// TwinCAT 3 PLC project PLC1
// Title: XPlanar Example Project
// Company: Beckhoff Automation LLC
// ProjectVersion: 1.0.0
// ProgramVersion: 3.1.4023.0
// libraries:
//   SPT Base Types, * (Beckhoff Automation LLC)
//   SPT Event Logger, * (Beckhoff Automation LLC)
//   SPT_XPlanar, * (Beckhoff Automation LLC)
//   Tc2_EtherCAT, * (Beckhoff Automation GmbH)
//   Tc2_Math, * (Beckhoff Automation GmbH)
//   Tc2_Standard, * (Beckhoff Automation GmbH)
//   Tc2_System, * (Beckhoff Automation GmbH)
//   Tc3_EventLogger, * (Beckhoff Automation GmbH)
//   Tc3_Module, * (Beckhoff Automation GmbH)
//   Tc3_PackML_V2, * (Beckhoff Automation GmbH)
//   Tc3_XPlanarUtility, * (Beckhoff Automation GmbH & Co. KG)
//   Tc3_Mc3PlanarMotion,newest,Beckhoff Automation GmbH
//   Tc3_Physics,newest,Beckhoff Automation GmbH
//   Tc3_XPlanarStandard,newest,Beckhoff Automation GmbH
//   VisuSymbols,3.5.10.0,System
// project tree:
//   DUTS/ ST_StationPosition.TcDUT, ST_VisMover.TcDUT, ST_VisStationData.TcDUT
//   / GlobalTextList.TcGTLO, MAIN.TcPOU, NextMinorStep.TcPOU, NextStep.TcPOU, PlcTask.TcTTO (not stored), StationList_TextList.TcTLO (not stored), Visualization Manager.TcVMO (not stored)
//   GVL/ GVL_Xplanar.TcGVL
//   Logic/Initialize/ FB_BasicInitialization.TcPOU, FB_MoverList.TcPOU
//   Machine/EquipmentModules/CustomStations/ FB_DecisionStation.TcPOU, FB_SpinStation.TcPOU
//   Machine/EquipmentModules/ FB_XPlanar_EM.TcPOU
//   Machine/ FB_Machine.TcPOU
//   Machine/VISUs/VisuOjects/ V_Control_Xplanar.TcVIS, V_MachineModule.TcVIS, V_Module.TcVIS (not stored), V_Mover.TcVIS (not stored), V_RotaryAxis.TcVIS (not stored), V_Station.TcVIS
//   Machine/VISUs/ V_Main.TcVIS
// real-time tasks:
//   TASK PlcTask: cycle T#10ms, priority 20, ADS port 350
//   TASK MC-Task (MET): cycle T#2ms, priority 7, ADS port 357
//   TASK MC-Task (MPT): cycle T#10ms, priority 8, ADS port 358
//   TASK Job Task: cycle default, priority 9
//   TASK XPlanar Task9: cycle T#250us, priority 1, ADS port 351
//   TASK XPlanar Task10: cycle T#250us, priority 2, ADS port 352
//   TASK XPlanar Task11: cycle T#250us, priority 3, ADS port 353
//   TASK XPlanar Task12: cycle T#250us, priority 4, ADS port 354
//   TASK XPlanar Task13: cycle T#250us, priority 5, ADS port 355
//   TASK XPlanar Task14: cycle T#250us, priority 6, ADS port 356
//   TASK XPlanar Task15: cycle T#250us, priority 10, ADS port 359
// variable links:
//   XPlanar MC Project/Axes/Mover4220_1 <-> TcCOM Objects/XPlanar/Mover4220_1
//     McToIo/STD <-> InputsFromNC3/NC3ToHW
//   XPlanar MC Project/Axes/Mover4220_10 <-> TcCOM Objects/XPlanar/Mover4220_10
//     McToIo/STD <-> InputsFromNC3/NC3ToHW
//   XPlanar MC Project/Axes/Mover4220_12 <-> TcCOM Objects/XPlanar/Mover4220_12
//     McToIo/STD <-> InputsFromNC3/NC3ToHW
//   XPlanar MC Project/Axes/Mover4220_13 <-> TcCOM Objects/XPlanar/Mover4220_13
//     IoToMc/STD <-> OutputsToNC3/HWToNC3
//   XPlanar MC Project/Axes/Mover4220_14 <-> TcCOM Objects/XPlanar/Mover4220_14
//     IoToMc/STD <-> OutputsToNC3/HWToNC3
//   XPlanar MC Project/Axes/Mover4220_15 <-> TcCOM Objects/XPlanar/Mover4220_15
//     IoToMc/STD <-> OutputsToNC3/HWToNC3
//     McToIo/STD <-> InputsFromNC3/NC3ToHW
//   XPlanar MC Project/Axes/Mover4220_17 <-> TcCOM Objects/XPlanar/Mover4220_17
//     IoToMc/STD <-> OutputsToNC3/HWToNC3
//     McToIo/STD <-> InputsFromNC3/NC3ToHW
//   XPlanar MC Project/Axes/Mover4220_18 <-> TcCOM Objects/XPlanar/Mover4220_18
//     IoToMc/STD <-> OutputsToNC3/HWToNC3
//     McToIo/STD <-> InputsFromNC3/NC3ToHW
//   XPlanar MC Project/Axes/Mover4220_19 <-> TcCOM Objects/XPlanar/Mover4220_19
//     McToIo/STD <-> InputsFromNC3/NC3ToHW
//   XPlanar MC Project/Axes/Mover4220_2 <-> TcCOM Objects/XPlanar/Mover4220_2
//     McToIo/STD <-> InputsFromNC3/NC3ToHW
//   XPlanar MC Project/Axes/Mover4220_3 <-> TcCOM Objects/XPlanar/Mover4220_3
//     IoToMc/STD <-> OutputsToNC3/HWToNC3
//   XPlanar MC Project/Axes/Mover4220_4 <-> TcCOM Objects/XPlanar/Mover4220_4
//     IoToMc/STD <-> OutputsToNC3/HWToNC3
//   XPlanar MC Project/Axes/Mover4220_5 <-> TcCOM Objects/XPlanar/Mover4220_5
//     IoToMc/STD <-> OutputsToNC3/HWToNC3
//     McToIo/STD <-> InputsFromNC3/NC3ToHW
//   XPlanar MC Project/Axes/Mover4220_6 <-> TcCOM Objects/XPlanar/Mover4220_6
//     McToIo/STD <-> InputsFromNC3/NC3ToHW
//   XPlanar MC Project/Axes/Mover4220_7 <-> TcCOM Objects/XPlanar/Mover4220_7
//     IoToMc/STD <-> OutputsToNC3/HWToNC3
//     McToIo/STD <-> InputsFromNC3/NC3ToHW
//   XPlanar MC Project/Axes/Mover4220_9 <-> TcCOM Objects/XPlanar/Mover4220_9
//     IoToMc/STD <-> OutputsToNC3/HWToNC3
//     McToIo/STD <-> InputsFromNC3/NC3ToHW
//   PLC1/PLC1 Instance <-> XPlanar MC Project/Axes/Mover4220_1
//     PlcTask Inputs/MAIN.Machine.XPlanar.Movers[1]._Mover.stMoverRef.MCTOPLC/ACT <-> McToPlc/ACT
//     PlcTask Inputs/MAIN.Machine.XPlanar.Movers[1]._Mover.stMoverRef.MCTOPLC/COORDMODE <-> McToPlc/COORDMODE
//     PlcTask Inputs/MAIN.Machine.XPlanar.Movers[1]._Mover.stMoverRef.MCTOPLC/SET <-> McToPlc/SET
//     PlcTask Inputs/MAIN.Machine.XPlanar.Movers[1]._Mover.stMoverRef.MCTOPLC/SETONTRACK <-> McToPlc/SETONTRACK
//     PlcTask Inputs/MAIN.Machine.XPlanar.Movers[1]._Mover.stMoverRef.MCTOPLC/STD <-> McToPlc/STD
//     PlcTask Outputs/MAIN.Machine.XPlanar.Movers[1]._Mover.stMoverRef.PLCTOMC/STD <-> PlcToMc/STD
//   PLC1/PLC1 Instance <-> XPlanar MC Project/Axes/Mover4220_10
//     PlcTask Inputs/MAIN.Machine.XPlanar.Movers[10]._Mover.stMoverRef.MCTOPLC/ACT <-> McToPlc/ACT
//     PlcTask Inputs/MAIN.Machine.XPlanar.Movers[10]._Mover.stMoverRef.MCTOPLC/COORDMODE <-> McToPlc/COORDMODE
//     PlcTask Inputs/MAIN.Machine.XPlanar.Movers[10]._Mover.stMoverRef.MCTOPLC/SET <-> McToPlc/SET
//     PlcTask Inputs/MAIN.Machine.XPlanar.Movers[10]._Mover.stMoverRef.MCTOPLC/SETONTRACK <-> McToPlc/SETONTRACK
//     PlcTask Inputs/MAIN.Machine.XPlanar.Movers[10]._Mover.stMoverRef.MCTOPLC/STD <-> McToPlc/STD
//     PlcTask Outputs/MAIN.Machine.XPlanar.Movers[10]._Mover.stMoverRef.PLCTOMC/STD <-> PlcToMc/STD
//   PLC1/PLC1 Instance <-> XPlanar MC Project/Axes/Mover4220_11
//     PlcTask Inputs/MAIN.Machine.XPlanar.Movers[11]._Mover.stMoverRef.MCTOPLC/ACT <-> McToPlc/ACT
//     PlcTask Inputs/MAIN.Machine.XPlanar.Movers[11]._Mover.stMoverRef.MCTOPLC/COORDMODE <-> McToPlc/COORDMODE
//     PlcTask Inputs/MAIN.Machine.XPlanar.Movers[11]._Mover.stMoverRef.MCTOPLC/SET <-> McToPlc/SET
//     PlcTask Inputs/MAIN.Machine.XPlanar.Movers[11]._Mover.stMoverRef.MCTOPLC/SETONTRACK <-> McToPlc/SETONTRACK
//     PlcTask Inputs/MAIN.Machine.XPlanar.Movers[11]._Mover.stMoverRef.MCTOPLC/STD <-> McToPlc/STD
//     PlcTask Outputs/MAIN.Machine.XPlanar.Movers[11]._Mover.stMoverRef.PLCTOMC/STD <-> PlcToMc/STD
//   PLC1/PLC1 Instance <-> XPlanar MC Project/Axes/Mover4220_12
//     PlcTask Inputs/MAIN.Machine.XPlanar.Movers[12]._Mover.stMoverRef.MCTOPLC/ACT <-> McToPlc/ACT
//     PlcTask Inputs/MAIN.Machine.XPlanar.Movers[12]._Mover.stMoverRef.MCTOPLC/COORDMODE <-> McToPlc/COORDMODE
//     PlcTask Inputs/MAIN.Machine.XPlanar.Movers[12]._Mover.stMoverRef.MCTOPLC/SET <-> McToPlc/SET
//     PlcTask Inputs/MAIN.Machine.XPlanar.Movers[12]._Mover.stMoverRef.MCTOPLC/SETONTRACK <-> McToPlc/SETONTRACK
//     PlcTask Inputs/MAIN.Machine.XPlanar.Movers[12]._Mover.stMoverRef.MCTOPLC/STD <-> McToPlc/STD
//     PlcTask Outputs/MAIN.Machine.XPlanar.Movers[12]._Mover.stMoverRef.PLCTOMC/STD <-> PlcToMc/STD
//   PLC1/PLC1 Instance <-> XPlanar MC Project/Axes/Mover4220_13
//     PlcTask Inputs/MAIN.Machine.XPlanar.Movers[13]._Mover.stMoverRef.MCTOPLC/ACT <-> McToPlc/ACT
//     PlcTask Inputs/MAIN.Machine.XPlanar.Movers[13]._Mover.stMoverRef.MCTOPLC/COORDMODE <-> McToPlc/COORDMODE
//     PlcTask Inputs/MAIN.Machine.XPlanar.Movers[13]._Mover.stMoverRef.MCTOPLC/SET <-> McToPlc/SET
//     PlcTask Inputs/MAIN.Machine.XPlanar.Movers[13]._Mover.stMoverRef.MCTOPLC/SETONTRACK <-> McToPlc/SETONTRACK
//     PlcTask Inputs/MAIN.Machine.XPlanar.Movers[13]._Mover.stMoverRef.MCTOPLC/STD <-> McToPlc/STD
//     PlcTask Outputs/MAIN.Machine.XPlanar.Movers[13]._Mover.stMoverRef.PLCTOMC/STD <-> PlcToMc/STD
//   PLC1/PLC1 Instance <-> XPlanar MC Project/Axes/Mover4220_14
//     PlcTask Inputs/MAIN.Machine.XPlanar.Movers[14]._Mover.stMoverRef.MCTOPLC/ACT <-> McToPlc/ACT
//     PlcTask Inputs/MAIN.Machine.XPlanar.Movers[14]._Mover.stMoverRef.MCTOPLC/COORDMODE <-> McToPlc/COORDMODE
//     PlcTask Inputs/MAIN.Machine.XPlanar.Movers[14]._Mover.stMoverRef.MCTOPLC/SET <-> McToPlc/SET
//     PlcTask Inputs/MAIN.Machine.XPlanar.Movers[14]._Mover.stMoverRef.MCTOPLC/SETONTRACK <-> McToPlc/SETONTRACK
//     PlcTask Inputs/MAIN.Machine.XPlanar.Movers[14]._Mover.stMoverRef.MCTOPLC/STD <-> McToPlc/STD
//     PlcTask Outputs/MAIN.Machine.XPlanar.Movers[14]._Mover.stMoverRef.PLCTOMC/STD <-> PlcToMc/STD
//   PLC1/PLC1 Instance <-> XPlanar MC Project/Axes/Mover4220_15
//     PlcTask Inputs/MAIN.Machine.XPlanar.Movers[15]._Mover.stMoverRef.MCTOPLC/ACT <-> McToPlc/ACT
//     PlcTask Inputs/MAIN.Machine.XPlanar.Movers[15]._Mover.stMoverRef.MCTOPLC/COORDMODE <-> McToPlc/COORDMODE
//     PlcTask Inputs/MAIN.Machine.XPlanar.Movers[15]._Mover.stMoverRef.MCTOPLC/SET <-> McToPlc/SET
//     PlcTask Inputs/MAIN.Machine.XPlanar.Movers[15]._Mover.stMoverRef.MCTOPLC/SETONTRACK <-> McToPlc/SETONTRACK
//     PlcTask Inputs/MAIN.Machine.XPlanar.Movers[15]._Mover.stMoverRef.MCTOPLC/STD <-> McToPlc/STD
//     PlcTask Outputs/MAIN.Machine.XPlanar.Movers[15]._Mover.stMoverRef.PLCTOMC/STD <-> PlcToMc/STD
//   PLC1/PLC1 Instance <-> XPlanar MC Project/Axes/Mover4220_16
//     PlcTask Inputs/MAIN.Machine.XPlanar.Movers[16]._Mover.stMoverRef.MCTOPLC/ACT <-> McToPlc/ACT
//     PlcTask Inputs/MAIN.Machine.XPlanar.Movers[16]._Mover.stMoverRef.MCTOPLC/COORDMODE <-> McToPlc/COORDMODE
//     PlcTask Inputs/MAIN.Machine.XPlanar.Movers[16]._Mover.stMoverRef.MCTOPLC/SET <-> McToPlc/SET
//     PlcTask Inputs/MAIN.Machine.XPlanar.Movers[16]._Mover.stMoverRef.MCTOPLC/SETONTRACK <-> McToPlc/SETONTRACK
//     PlcTask Inputs/MAIN.Machine.XPlanar.Movers[16]._Mover.stMoverRef.MCTOPLC/STD <-> McToPlc/STD
//     PlcTask Outputs/MAIN.Machine.XPlanar.Movers[16]._Mover.stMoverRef.PLCTOMC/STD <-> PlcToMc/STD
//   PLC1/PLC1 Instance <-> XPlanar MC Project/Axes/Mover4220_17
//     PlcTask Inputs/MAIN.Machine.XPlanar.Movers[17]._Mover.stMoverRef.MCTOPLC/ACT <-> McToPlc/ACT
//     PlcTask Inputs/MAIN.Machine.XPlanar.Movers[17]._Mover.stMoverRef.MCTOPLC/COORDMODE <-> McToPlc/COORDMODE
//     PlcTask Inputs/MAIN.Machine.XPlanar.Movers[17]._Mover.stMoverRef.MCTOPLC/SET <-> McToPlc/SET
//     PlcTask Inputs/MAIN.Machine.XPlanar.Movers[17]._Mover.stMoverRef.MCTOPLC/SETONTRACK <-> McToPlc/SETONTRACK
//     PlcTask Inputs/MAIN.Machine.XPlanar.Movers[17]._Mover.stMoverRef.MCTOPLC/STD <-> McToPlc/STD
//     PlcTask Outputs/MAIN.Machine.XPlanar.Movers[17]._Mover.stMoverRef.PLCTOMC/STD <-> PlcToMc/STD
//   PLC1/PLC1 Instance <-> XPlanar MC Project/Axes/Mover4220_18
//     PlcTask Inputs/MAIN.Machine.XPlanar.Movers[18]._Mover.stMoverRef.MCTOPLC/ACT <-> McToPlc/ACT
//     PlcTask Inputs/MAIN.Machine.XPlanar.Movers[18]._Mover.stMoverRef.MCTOPLC/COORDMODE <-> McToPlc/COORDMODE
//     PlcTask Inputs/MAIN.Machine.XPlanar.Movers[18]._Mover.stMoverRef.MCTOPLC/SET <-> McToPlc/SET
//     PlcTask Inputs/MAIN.Machine.XPlanar.Movers[18]._Mover.stMoverRef.MCTOPLC/SETONTRACK <-> McToPlc/SETONTRACK
//     PlcTask Inputs/MAIN.Machine.XPlanar.Movers[18]._Mover.stMoverRef.MCTOPLC/STD <-> McToPlc/STD
//     PlcTask Outputs/MAIN.Machine.XPlanar.Movers[18]._Mover.stMoverRef.PLCTOMC/STD <-> PlcToMc/STD
//   PLC1/PLC1 Instance <-> XPlanar MC Project/Axes/Mover4220_19
//     PlcTask Inputs/MAIN.Machine.XPlanar.Movers[19]._Mover.stMoverRef.MCTOPLC/ACT <-> McToPlc/ACT
//     PlcTask Inputs/MAIN.Machine.XPlanar.Movers[19]._Mover.stMoverRef.MCTOPLC/COORDMODE <-> McToPlc/COORDMODE
//     PlcTask Inputs/MAIN.Machine.XPlanar.Movers[19]._Mover.stMoverRef.MCTOPLC/SET <-> McToPlc/SET
//     PlcTask Inputs/MAIN.Machine.XPlanar.Movers[19]._Mover.stMoverRef.MCTOPLC/SETONTRACK <-> McToPlc/SETONTRACK
//     PlcTask Inputs/MAIN.Machine.XPlanar.Movers[19]._Mover.stMoverRef.MCTOPLC/STD <-> McToPlc/STD
//     PlcTask Outputs/MAIN.Machine.XPlanar.Movers[19]._Mover.stMoverRef.PLCTOMC/STD <-> PlcToMc/STD
//   PLC1/PLC1 Instance <-> XPlanar MC Project/Axes/Mover4220_2
//     PlcTask Inputs/MAIN.Machine.XPlanar.Movers[2]._Mover.stMoverRef.MCTOPLC/ACT <-> McToPlc/ACT
//     PlcTask Inputs/MAIN.Machine.XPlanar.Movers[2]._Mover.stMoverRef.MCTOPLC/COORDMODE <-> McToPlc/COORDMODE
//     PlcTask Inputs/MAIN.Machine.XPlanar.Movers[2]._Mover.stMoverRef.MCTOPLC/SET <-> McToPlc/SET
//     PlcTask Inputs/MAIN.Machine.XPlanar.Movers[2]._Mover.stMoverRef.MCTOPLC/SETONTRACK <-> McToPlc/SETONTRACK
//     PlcTask Inputs/MAIN.Machine.XPlanar.Movers[2]._Mover.stMoverRef.MCTOPLC/STD <-> McToPlc/STD
//     PlcTask Outputs/MAIN.Machine.XPlanar.Movers[2]._Mover.stMoverRef.PLCTOMC/STD <-> PlcToMc/STD
//   PLC1/PLC1 Instance <-> XPlanar MC Project/Axes/Mover4220_3
//     PlcTask Inputs/MAIN.Machine.XPlanar.Movers[3]._Mover.stMoverRef.MCTOPLC/ACT <-> McToPlc/ACT
//     PlcTask Inputs/MAIN.Machine.XPlanar.Movers[3]._Mover.stMoverRef.MCTOPLC/COORDMODE <-> McToPlc/COORDMODE
//     PlcTask Inputs/MAIN.Machine.XPlanar.Movers[3]._Mover.stMoverRef.MCTOPLC/SET <-> McToPlc/SET
//     PlcTask Inputs/MAIN.Machine.XPlanar.Movers[3]._Mover.stMoverRef.MCTOPLC/SETONTRACK <-> McToPlc/SETONTRACK
//     PlcTask Inputs/MAIN.Machine.XPlanar.Movers[3]._Mover.stMoverRef.MCTOPLC/STD <-> McToPlc/STD
//     PlcTask Outputs/MAIN.Machine.XPlanar.Movers[3]._Mover.stMoverRef.PLCTOMC/STD <-> PlcToMc/STD
//   PLC1/PLC1 Instance <-> XPlanar MC Project/Axes/Mover4220_4
//     PlcTask Inputs/MAIN.Machine.XPlanar.Movers[4]._Mover.stMoverRef.MCTOPLC/ACT <-> McToPlc/ACT
//     PlcTask Inputs/MAIN.Machine.XPlanar.Movers[4]._Mover.stMoverRef.MCTOPLC/COORDMODE <-> McToPlc/COORDMODE
//     PlcTask Inputs/MAIN.Machine.XPlanar.Movers[4]._Mover.stMoverRef.MCTOPLC/SET <-> McToPlc/SET
//     PlcTask Inputs/MAIN.Machine.XPlanar.Movers[4]._Mover.stMoverRef.MCTOPLC/SETONTRACK <-> McToPlc/SETONTRACK
//     PlcTask Inputs/MAIN.Machine.XPlanar.Movers[4]._Mover.stMoverRef.MCTOPLC/STD <-> McToPlc/STD
//     PlcTask Outputs/MAIN.Machine.XPlanar.Movers[4]._Mover.stMoverRef.PLCTOMC/STD <-> PlcToMc/STD
//   PLC1/PLC1 Instance <-> XPlanar MC Project/Axes/Mover4220_5
//     PlcTask Inputs/MAIN.Machine.XPlanar.Movers[5]._Mover.stMoverRef.MCTOPLC/ACT <-> McToPlc/ACT
//     PlcTask Inputs/MAIN.Machine.XPlanar.Movers[5]._Mover.stMoverRef.MCTOPLC/COORDMODE <-> McToPlc/COORDMODE
//     PlcTask Inputs/MAIN.Machine.XPlanar.Movers[5]._Mover.stMoverRef.MCTOPLC/SET <-> McToPlc/SET
//     PlcTask Inputs/MAIN.Machine.XPlanar.Movers[5]._Mover.stMoverRef.MCTOPLC/SETONTRACK <-> McToPlc/SETONTRACK
//     PlcTask Inputs/MAIN.Machine.XPlanar.Movers[5]._Mover.stMoverRef.MCTOPLC/STD <-> McToPlc/STD
//     PlcTask Outputs/MAIN.Machine.XPlanar.Movers[5]._Mover.stMoverRef.PLCTOMC/STD <-> PlcToMc/STD
//   PLC1/PLC1 Instance <-> XPlanar MC Project/Axes/Mover4220_6
//     PlcTask Inputs/MAIN.Machine.XPlanar.Movers[6]._Mover.stMoverRef.MCTOPLC/ACT <-> McToPlc/ACT
//     PlcTask Inputs/MAIN.Machine.XPlanar.Movers[6]._Mover.stMoverRef.MCTOPLC/COORDMODE <-> McToPlc/COORDMODE
//     PlcTask Inputs/MAIN.Machine.XPlanar.Movers[6]._Mover.stMoverRef.MCTOPLC/SET <-> McToPlc/SET
//     PlcTask Inputs/MAIN.Machine.XPlanar.Movers[6]._Mover.stMoverRef.MCTOPLC/SETONTRACK <-> McToPlc/SETONTRACK
//     PlcTask Inputs/MAIN.Machine.XPlanar.Movers[6]._Mover.stMoverRef.MCTOPLC/STD <-> McToPlc/STD
//     PlcTask Outputs/MAIN.Machine.XPlanar.Movers[6]._Mover.stMoverRef.PLCTOMC/STD <-> PlcToMc/STD
//   PLC1/PLC1 Instance <-> XPlanar MC Project/Axes/Mover4220_7
//     PlcTask Inputs/MAIN.Machine.XPlanar.Movers[7]._Mover.stMoverRef.MCTOPLC/ACT <-> McToPlc/ACT
//     PlcTask Inputs/MAIN.Machine.XPlanar.Movers[7]._Mover.stMoverRef.MCTOPLC/COORDMODE <-> McToPlc/COORDMODE
//     PlcTask Inputs/MAIN.Machine.XPlanar.Movers[7]._Mover.stMoverRef.MCTOPLC/SET <-> McToPlc/SET
//     PlcTask Inputs/MAIN.Machine.XPlanar.Movers[7]._Mover.stMoverRef.MCTOPLC/SETONTRACK <-> McToPlc/SETONTRACK
//     PlcTask Inputs/MAIN.Machine.XPlanar.Movers[7]._Mover.stMoverRef.MCTOPLC/STD <-> McToPlc/STD
//     PlcTask Outputs/MAIN.Machine.XPlanar.Movers[7]._Mover.stMoverRef.PLCTOMC/STD <-> PlcToMc/STD
//   PLC1/PLC1 Instance <-> XPlanar MC Project/Axes/Mover4220_8
//     PlcTask Inputs/MAIN.Machine.XPlanar.Movers[8]._Mover.stMoverRef.MCTOPLC/ACT <-> McToPlc/ACT
//     PlcTask Inputs/MAIN.Machine.XPlanar.Movers[8]._Mover.stMoverRef.MCTOPLC/COORDMODE <-> McToPlc/COORDMODE
//     PlcTask Inputs/MAIN.Machine.XPlanar.Movers[8]._Mover.stMoverRef.MCTOPLC/SET <-> McToPlc/SET
//     PlcTask Inputs/MAIN.Machine.XPlanar.Movers[8]._Mover.stMoverRef.MCTOPLC/SETONTRACK <-> McToPlc/SETONTRACK
//     PlcTask Inputs/MAIN.Machine.XPlanar.Movers[8]._Mover.stMoverRef.MCTOPLC/STD <-> McToPlc/STD
//     PlcTask Outputs/MAIN.Machine.XPlanar.Movers[8]._Mover.stMoverRef.PLCTOMC/STD <-> PlcToMc/STD
//   PLC1/PLC1 Instance <-> XPlanar MC Project/Axes/Mover4220_9
//     PlcTask Inputs/MAIN.Machine.XPlanar.Movers[9]._Mover.stMoverRef.MCTOPLC/ACT <-> McToPlc/ACT
//     PlcTask Inputs/MAIN.Machine.XPlanar.Movers[9]._Mover.stMoverRef.MCTOPLC/COORDMODE <-> McToPlc/COORDMODE
//     PlcTask Inputs/MAIN.Machine.XPlanar.Movers[9]._Mover.stMoverRef.MCTOPLC/SET <-> McToPlc/SET
//     PlcTask Inputs/MAIN.Machine.XPlanar.Movers[9]._Mover.stMoverRef.MCTOPLC/SETONTRACK <-> McToPlc/SETONTRACK
//     PlcTask Inputs/MAIN.Machine.XPlanar.Movers[9]._Mover.stMoverRef.MCTOPLC/STD <-> McToPlc/STD
//     PlcTask Outputs/MAIN.Machine.XPlanar.Movers[9]._Mover.stMoverRef.PLCTOMC/STD <-> PlcToMc/STD
//   PLC1/PLC1 Instance <-> XPlanar MC Project/Groups/Environment
//     PlcTask Inputs/MAIN.Machine.XPlanar.XPlanarTable.XPlanarSystem.environment.MCTOPLC_STD <-> McToPlc/STD
//   PLC1/PLC1 Instance <-> XPlanar MC Project/Groups/Group3 (Planar Track)
//     PlcTask Inputs/MAIN.Machine.XPlanar.Tracks[1].TrackStandard.stTrackRef.MCTOPLC_STD <-> McToPlc/STD
//   PLC1/PLC1 Instance <-> XPlanar MC Project/Groups/Group4 (Planar Track)
//     PlcTask Inputs/MAIN.Machine.XPlanar.Tracks[2].TrackStandard.stTrackRef.MCTOPLC_STD <-> McToPlc/STD
//   PLC1/PLC1 Instance <-> XPlanar MC Project/Groups/Group5 (Planar Track)
//     PlcTask Inputs/MAIN.Machine.XPlanar.Tracks[3].TrackStandard.stTrackRef.MCTOPLC_STD <-> McToPlc/STD
//   PLC1/PLC1 Instance <-> XPlanar MC Project/Groups/Group6 (Planar Track)
//     PlcTask Inputs/MAIN.Machine.XPlanar.Tracks[4].TrackStandard.stTrackRef.MCTOPLC_STD <-> McToPlc/STD
//   PLC1/PLC1 Instance <-> XPlanar MC Project/Groups/XPlanar
//     PlcTask Inputs/MAIN.Machine.XPlanar.XPlanarTable.XPlanarSystem.group.MCTOPLC_STD <-> McToPlc/STD
//   TcCOM Objects/XPlanar/Mover4220_1 <-> XPlanar MC Project/Axes/Mover4220_1
//     OutputsToNC3/HWToNC3 <-> IoToMc/STD
//   TcCOM Objects/XPlanar/Mover4220_10 <-> XPlanar MC Project/Axes/Mover4220_10
//     OutputsToNC3/HWToNC3 <-> IoToMc/STD
//   TcCOM Objects/XPlanar/Mover4220_11 <-> XPlanar MC Project/Axes/Mover4220_11
//     InputsFromNC3/NC3ToHW <-> McToIo/STD
//     OutputsToNC3/HWToNC3 <-> IoToMc/STD
//   TcCOM Objects/XPlanar/Mover4220_12 <-> XPlanar MC Project/Axes/Mover4220_12
//     OutputsToNC3/HWToNC3 <-> IoToMc/STD
//   TcCOM Objects/XPlanar/Mover4220_13 <-> XPlanar MC Project/Axes/Mover4220_13
//     InputsFromNC3/NC3ToHW <-> McToIo/STD
//   TcCOM Objects/XPlanar/Mover4220_14 <-> XPlanar MC Project/Axes/Mover4220_14
//     InputsFromNC3/NC3ToHW <-> McToIo/STD
//   TcCOM Objects/XPlanar/Mover4220_16 <-> XPlanar MC Project/Axes/Mover4220_16
//     InputsFromNC3/NC3ToHW <-> McToIo/STD
//     OutputsToNC3/HWToNC3 <-> IoToMc/STD
//   TcCOM Objects/XPlanar/Mover4220_19 <-> XPlanar MC Project/Axes/Mover4220_19
//     OutputsToNC3/HWToNC3 <-> IoToMc/STD
//   TcCOM Objects/XPlanar/Mover4220_2 <-> XPlanar MC Project/Axes/Mover4220_2
//     OutputsToNC3/HWToNC3 <-> IoToMc/STD
//   TcCOM Objects/XPlanar/Mover4220_3 <-> XPlanar MC Project/Axes/Mover4220_3
//     InputsFromNC3/NC3ToHW <-> McToIo/STD
//   TcCOM Objects/XPlanar/Mover4220_4 <-> XPlanar MC Project/Axes/Mover4220_4
//     InputsFromNC3/NC3ToHW <-> McToIo/STD
//   TcCOM Objects/XPlanar/Mover4220_6 <-> XPlanar MC Project/Axes/Mover4220_6
//     OutputsToNC3/HWToNC3 <-> IoToMc/STD
//   TcCOM Objects/XPlanar/Mover4220_8 <-> XPlanar MC Project/Axes/Mover4220_8
//     InputsFromNC3/NC3ToHW <-> McToIo/STD
//     OutputsToNC3/HWToNC3 <-> IoToMc/STD

// ---- DUTS/ST_StationPosition.TcDUT
TYPE ST_StationPosition :
STRUCT
	fpositionX			: LREAL;
	fpositionY			: LREAL;
END_STRUCT
END_TYPE

// ---- DUTS/ST_VisMover.TcDUT
TYPE ST_VisMover :
STRUCT
	fPosition_X	: LREAL;
	fPosition_Y 	: LREAL;
	fPosition_Z	: LREAL;
	fPosition_A 	: LREAL;
	fPosition_B	: LREAL;
	fPosition_C	: LREAL;
	
END_STRUCT
END_TYPE

// ---- DUTS/ST_VisStationData.TcDUT
TYPE ST_VisStationData :

STRUCT
	
	bInit		: BOOL;
	fPosition_X	: LREAL;
	fPosition_Y : LREAL;

END_STRUCT

END_TYPE

// ---- GVL/GVL_Xplanar.TcGVL
VAR_GLOBAL
	CONSTANT
		MAX_STATION_NUMBER		: UDINT :=3;
		MAX_MOVERS							: UDINT := 19;
END_VAR
VAR_GLOBAL
//	MAX_MOVERS		: UDINT:=Tc3_XPlanarStandard.Params_XPlanar.moverCount;
//	MAX_TRACKS		: UDINT:=Tc3_XPlanarStandard.Params_XPlanar.maxTrackCount;

	stStationPos						:ARRAY[1..MAX_STATION_NUMBER] OF ST_StationPosition;
	stStationVis						:ARRAY[1..MAX_STATION_NUMBER] OF ST_VisStationData;
	stMoverVis						:ARRAY[1..Tc3_XPlanarStandard.Params_XPlanar.moverCount] OF ST_VisMover;
	
	SetInitVelo					: LREAL:=500;
	SetInitAccDec				: LREAL:=1000;
	SetInitJerk						: LREAL:=5000;
	
END_VAR

// ---- Logic/Initialize/FB_BasicInitialization.TcPOU
FUNCTION_BLOCK FB_BasicInitialization
VAR_INPUT
	bExcute								: BOOL;
	nSizeOfMover					: INT;
	aLocationOfArea				: ARRAY[1..4,1..2] OF REAL;	
	ipMover								: ARRAY [0..Tc3_XPlanarStandard.Params_XPlanar.moverCount] OF I_XPlanarMover;//I_Mover;
	bReset								: BOOL;	
	
END_VAR
VAR_OUTPUT
	Busy									: BOOL;
	Done									: BOOL;
	Error									: BOOL;
	ErrorCode							: WSTRING;
	
	
	
END_VAR
VAR
	bFlagAuto						: BOOL;
	bFlagManual         		: BOOL;
	nState								: INT;
	bStart								: BOOL;
	nZoneColumn				: INT;
	nZoneRow						: INT;	
	aTable							: ARRAY[1..20]OF INT;
	aInitialPoint					: ARRAY[1..20,1..2] OF REAL;
	fZoneLengthX				: REAL;
	fZoneLengthY				: REAL;
	SortingState						:INT;	
	MovingState						:INT;	
	bDone 					: BOOL;
	fbMoverSortList				:ARRAY[1..10] OF FB_MoverList;	
	nCounterX							:ARRAY[1..20] OF INT;									//mover number in every zone
//	nTileRowCount								: INT :=3;
//	nTileColumnCount						: INT :=4;
//	MOVER_LENGTH							: REAL:=156;	
//	fTileLengthX									: LREAL :=240*nTileColumnCount;
//	fTileLengthY									: LREAL :=240*nTileRowCount;
END_VAR
VAR_IN_OUT
	aManualPos					: ARRAY [*,*] OF REAL;
END_VAR

IF bExcute = TRUE THEN
	IF nSizeOfMover <>115 AND nSizeOfMover <> 155 AND nSizeOfMover <> 235 THEN
		Error  := TRUE;
		ErrorCode := "Mover size is not correct";
	ELSE
		bStart := bExcute AND NOT Error ;
	END_IF	
END_IF

IF bStart THEN
	CASE nState OF
		
	0:
		IF M_CalculateArea(nSizeOfMover:=nSizeOfMover,aLocationOfArea:=aLocationOfArea,nZoneColumn=>nZoneColumn,nZoneRow=>nZoneRow,fZoneLengthX=>fZoneLengthX,fZoneLengthY=>fZoneLengthY) = TRUE THEN
				Busy := TRUE;
				Error  := FALSE;
				ErrorCode := "";
				nState := 10;
			ELSE
				Error  := TRUE;
				ErrorCode := "Area is not correct";			
				nState := 99;	
		END_IF 
		
	10:
		IF M_JudgePoint(aManualPos:=aManualPos) = TRUE THEN
				Busy := TRUE;
				Error  := FALSE;
				ErrorCode := "";
				nState := 20;
			ELSE
				Error  := TRUE;
				ErrorCode := "Point is not correct";			
				nState := 99;	
		END_IF				
	
	20:
		IF M_CreateTable(nSizeOfMover:=nSizeOfMover,nZoneColumn:=nZoneColumn,nZoneRow:=nZoneRow,aLocationOfArea:=aLocationOfArea,fZoneLengthY:=fZoneLengthY,aManualPos:=aManualPos,aTable=>aTable) = TRUE THEN
				Busy := TRUE;
				Error  := FALSE;
				ErrorCode := "";
				nState := 30;
			ELSE
				Error  := TRUE;
				ErrorCode := "Position is not correct";	
				nState := 99;				
		END_IF 	
	
	
	30:
				IF M_MoverSorting(nSizeOfMover:=nSizeOfMover,nZoneColumn:=nZoneColumn,nZoneRow:=nZoneRow,aTable:=aTable,fZoneLengthX:=fZoneLengthX,fZoneLengthY:=fZoneLengthY) = TRUE THEN
					Busy := TRUE;		
					Done := FALSE;		
					nState := 40;	
				END_IF
				
	40:
				IF M_MoveToInitialPos(aManualPos:=aManualPos) = TRUE THEN
//					Busy := FALSE;		
//					Done := TRUE;		
					nState := 100;	
				END_IF		

	END_CASE
END_IF

IF bReset THEN
	THIS^.FB_init(TRUE,TRUE);
END_IF

METHOD FB_init : BOOL
VAR_INPUT
	bInitRetains : BOOL; // if TRUE, the retain variables are initialized (warm start / cold start)
	bInCopyCode : BOOL;  // if TRUE, the instance afterwards gets moved into the copy code (online change)
END_VAR
END_METHOD

METHOD M_CalculateArea : BOOL
VAR_INPUT
		nSizeOfMover					: INT;
		aLocationOfArea				: ARRAY[1..4,1..2] OF REAL;	
END_VAR
VAR_OUTPUT
	nZoneRow							: INT;
	nZoneColumn					: INT;
	fZoneLengthX					: REAL;
	fZoneLengthY					: REAL;
END_VAR
VAR_INST
	fRegionalArea					: REAL;	
END_VAR
IF aLocationOfArea[1,1] >= 0 AND aLocationOfArea[1,2] >= 0 AND aLocationOfArea[2,1] >= 0 AND aLocationOfArea[2,2] >= 0 AND
	aLocationOfArea[3,1] >= 0 AND aLocationOfArea[3,2] >= 0 AND aLocationOfArea[4,1] >= 0 AND aLocationOfArea[4,2] >= 0 AND
	aLocationOfArea[2,1] > aLocationOfArea[1,1] AND aLocationOfArea[4,1] > aLocationOfArea[3,1] AND
	aLocationOfArea[2,2] > aLocationOfArea[4,2] AND aLocationOfArea[1,2] > aLocationOfArea[3,2] AND
	aLocationOfArea[2,2] = aLocationOfArea[1,2] AND aLocationOfArea[4,2] = aLocationOfArea[3,2] AND
	aLocationOfArea[1,1] = aLocationOfArea[3,1] AND aLocationOfArea[2,1] = aLocationOfArea[4,1] THEN
	fZoneLengthX := aLocationOfArea[2,1] - aLocationOfArea[1,1];
	fZoneLengthY := aLocationOfArea[2,2] - aLocationOfArea[4,2];
	fRegionalArea := fZoneLengthX*fZoneLengthY;
	IF nSizeOfMover*nSizeOfMover > fRegionalArea/4 THEN
		    M_CalculateArea :=FALSE;
		ELSE
			nZoneRow :=LREAL_TO_INT(FLOOR(fZoneLengthY/INT_TO_REAL(nSizeOfMover+5)));
			nZoneColumn :=LREAL_TO_INT(FLOOR(fZoneLengthX/INT_TO_REAL(nSizeOfMover+5)));			
	END_IF
END_IF

IF nZoneColumn > 0 AND nZoneRow >0 THEN
	M_CalculateArea := TRUE;
END_IF
END_METHOD

METHOD M_CreateTable : BOOL
VAR_INPUT
		nSizeOfMover					: INT;
		aLocationOfArea				: ARRAY[1..4,1..2] OF REAL;	
		nZoneColumn					: INT;
		nZoneRow							: INT;	
		fZoneLengthY					: REAL;
END_VAR
VAR_OUTPUT
//	aMoverIndexInArea				: ARRAY[1..20] OF INT;
	aTable									: ARRAY[1..20] OF INT;
END_VAR
VAR_IN_OUT
	aManualPos							: ARRAY [*,*] OF REAL;

END_VAR

VAR
	i										: INT;
	nCounter						: INT;
	nCounter2						: INT;
	j										: INT;
	k										: INT;
    nAL1								: INT 		:= DINT_TO_INT(LOWER_BOUND(aManualPos, 1));						//row
    nAU1								: INT 		:= DINT_TO_INT(UPPER_BOUND(aManualPos, 1));
    nAL2								: INT 		:= DINT_TO_INT(LOWER_BOUND(aManualPos, 2));						//col
    nAU2								: INT 		:= DINT_TO_INT(UPPER_BOUND(aManualPos, 2));
	nRemainder					:INT;
	fdistance						: REAL;
	ftemp								: REAL;
	nArrayIsEmpty				: BOOL;
	aTemp							: ARRAY[1..20,1..2] OF REAL;
	aInitialPoint					: ARRAY [1..20,1..2] OF REAL;
END_VAR
FOR  i := 1 TO TO_INT(Tc3_XPlanarStandard.Params_XPlanar.moverCount) DO
	IF ipMover[i].std.P_ActPosition.x > aLocationOfArea[1,1] AND ipMover[i].std.P_ActPosition.y < aLocationOfArea[1,2] AND
		ipMover[i].std.P_ActPosition.x < aLocationOfArea[4,1] AND ipMover[i].std.P_ActPosition.y > aLocationOfArea[4,2] THEN
		nCounter := nCounter + 1;
//		j := j + 1;
//		aMoverIndexInArea[j] := i;
	END_IF
END_FOR

FOR i := 1 TO nAU1 DO
	FOR j := 1 TO nAU2 DO
		IF aManualPos[i,j] <> 0 THEN
			nArrayIsEmpty:= TRUE;	
		END_IF
	END_FOR
END_FOR


IF nAU1 =0 OR nAU2  = 0  OR nArrayIsEmpty = FALSE THEN
		IF nCounter <> 0 THEN																															// auto mode
			
		
			k := nCounter/nZoneRow;
			nRemainder := nCounter MOD nZoneRow;
			IF k >= 1 THEN
				FOR i:=1 TO nZoneRow DO
					aTable[i] := k;		
				END_FOR	
				FOR i:=1 TO nZoneRow DO
					IF nRemainder > 0 THEN
						aTable[i] := aTable[i] + 1;				
						nRemainder := nRemainder-1;
					END_IF
				END_FOR	

				ELSE
					FOR i:=1 TO nRemainder DO
						aTable[i] := 1;	
					END_FOR				
			END_IF
		
			M_CreateTable := TRUE;		
		
		END_IF

	ELSE																																							// manual mode
		IF nCounter <> 0 THEN//AND nCounter = nAU1 THEN	
   			FOR i:=1 TO nAU1 DO
				FOR j:=1 TO 2 DO
					aInitialPoint[i,j]:=aManualPos[i,j];				
				END_FOR
			END_FOR
   			FOR i:=1 TO nAU1 DO		
				FOR j:=1 TO nAU1 DO		
						fdistance:=SQRT((aLocationOfArea[1,1]-aInitialPoint[j,1])*(aLocationOfArea[1,1]-aInitialPoint[j,1]) + (aLocationOfArea[1,2]-aInitialPoint[j,2])*(aLocationOfArea[1,2]-aInitialPoint[j,2]));
						IF fdistance < ftemp THEN
							ftemp := fdistance;
							aTemp[j,1] := aInitialPoint[j,1];
							aTemp[j,2] := aInitialPoint[j,2];	
							aInitialPoint[j,1] := aInitialPoint[j+1,1];
							aInitialPoint[j,2] := aInitialPoint[j+1,2];	
							aInitialPoint[j+1,1] := aTemp[j,1];
							aInitialPoint[j+1,2] := aTemp[j,2];							
						END_IF
				END_FOR
			END_FOR
	
			FOR i := 1 TO nZoneRow DO
				FOR j := 1 TO 2 DO
					aManualPos[i,j]:=	aInitialPoint[i,j];			
				END_FOR
			END_FOR
		
			FOR i := 1 TO nZoneRow DO
				FOR j := 1 TO nCounter DO
					IF aInitialPoint[j,2] <=  fZoneLengthY*(nZoneRow+1-i)/nZoneRow AND aInitialPoint[j,2] >  fZoneLengthY*(nZoneRow-i)/nZoneRow THEN
						aTable[i] := aTable[i] + 1;		
					END_IF					
				END_FOR
			END_FOR
		
			M_CreateTable := TRUE;			
		END_IF
END_IF
END_METHOD

METHOD M_JudgePoint : BOOL
VAR_INPUT
END_VAR
VAR_IN_OUT
	aManualPos							: ARRAY [*,*] OF REAL;
END_VAR

VAR
	nAL1								: INT 		:= DINT_TO_INT(LOWER_BOUND(aManualPos, 1));						//row
    nAU1								: INT 		:= DINT_TO_INT(UPPER_BOUND(aManualPos, 1));
    nAL2								: INT 		:= DINT_TO_INT(LOWER_BOUND(aManualPos, 2));						//col
    nAU2								: INT 		:= DINT_TO_INT(UPPER_BOUND(aManualPos, 2));
	i,j,k									: INT;
	fDis									: REAL;
	bJudge1							: BOOL;
	bJudge2							: BOOL;
END_VAR
//Judge whether  the aManualPos points is appropriate and whether the boundary will be touched
bJudge1 := TRUE;
bJudge2 := TRUE;
FOR i := 1 TO nAU1-1 DO
		bJudge1 := bJudge1 AND (aManualPos[i,1] - TO_REAL(nSizeOfMover)/2.0 >=1) AND (aManualPos[i,2] - TO_REAL(nSizeOfMover)/2.0 >=1 );
		FOR j := i TO nAU1-1 DO
			fDis := SQRT((aManualPos[j,1] -  aManualPos[j+1,1])*(aManualPos[j,1] -  aManualPos[j+1,1]) + (aManualPos[j,2] -  aManualPos[j+1,2])*(aManualPos[j,2] -  aManualPos[j+1,2]));
			bJudge2 := bJudge2 AND (fDis > nSizeOfMover + 7 );
		END_FOR
END_FOR

IF bJudge1 AND bJudge2 THEN
	M_JudgePoint := TRUE;
END_IF
END_METHOD

METHOD M_MoverSorting : BOOL
VAR_INPUT
	nSizeOfMover				: INT;
	nZoneColumn				: INT;
	nZoneRow						: INT;	
	aTable							: ARRAY[1..20]OF INT;
	fZoneLengthX					: REAL;
	fZoneLengthY					: REAL;
END_VAR
VAR_INST
	i,j,k							:INT;
	InitList					:FB_MoverList;
	nSorting					: ARRAY [1..20] OF INT;
	
	fTileLengthX									: LREAL ;
	fTileLengthY									: LREAL ;
	
	nMoverIndex					:INT ;
	Xpoint								:LREAL;
	Ypoint								:LREAL;
	nZoneCounter					:INT;																	// zone number
	nCounterMem					:ARRAY[1..10] OF INT;									//mover number difference expected
	nMoverIistInZone			: ARRAY[0..Tc3_XPlanarStandard.Params_XPlanar.moverCount] OF INT;

	bGet									: BOOL;
	nGet									:INT;
	bGive									: BOOL;
	nGive									:INT;	
	bFirstGive							: BOOL;
	bFirstGet							: BOOL;
	nMAX									:INT;
	nMAXTemp						: INT;
	nPos									:INT;
	fLengthGive						:LREAL;
	fLengthY							:LREAL;
	fLengthGet						:LREAL;
	Pos										:PositionXYC;

	InitVelo							:LREAL;
	InitAcc,InitDec				:LREAL;
	InitJerk							:LREAL;

END_VAR
	InitVelo:=SetInitVelo;
	InitAcc:=SetInitAccDec;
	InitDec:=SetInitAccDec;
	InitJerk:=SetInitJerk;

IF bReset THEN
	SortingState := 0;
	nMoverIndex :=0;
	nZoneCounter:=0;
END_IF

CASE SortingState OF
	0:
		FOR i:=1 TO TO_INT(Tc3_XPlanarStandard.Params_XPlanar.moverCount) DO 
			InitList.M_AddToList(i);
		END_FOR
		SortingState:=1;
	1:
		fTileLengthY := TO_LREAL(fZoneLengthY);
		fTileLengthX := TO_LREAL(fZoneLengthX);		
		FOR i := 1 TO 20 DO
			nSorting[i] := aTable[i];
		END_FOR
		SortingState:=10;
	10:
		IF InitList.List[0]>0 THEN 
			nMoverIndex:=0;
			memset(ADR(nCounterX),0,SIZEOF(nCounterX));
			k:=1;
			SortingState:=20;
		END_IF
		
		
///////////////////////************Movers within each zone move to the top of the zone in turn*************/////////////////////////////
	20:
		IF nMoverIndex<Tc3_XPlanarStandard.Params_XPlanar.moverCount THEN 
			nMoverIndex:=nMoverIndex+1;
			SortingState:=30;
		ELSE
			SortingState:=60;
		END_IF
	30:
		Xpoint:=ipMover[nMoverIndex].std.P_SetPosition.x;
		Ypoint:=ipMover[nMoverIndex].std.P_SetPosition.y;
		IF Ypoint <= fTileLengthY*(nZoneRow-nZoneCounter)/nZoneRow-TO_REAL(nSizeOfMover)/2.0
			AND Ypoint >= fTileLengthY*(nZoneRow-nZoneCounter-1)/nZoneRow-TO_REAL(nSizeOfMover)/2.0 THEN
//			AND F_CheckMoverCanMove(nMoverIndex,Xpoint,Ypoint,ipMover) THEN
			SortingState:=40;			
		ELSE
			SortingState:=20;
		END_IF	

	40:
		Pos.SetValuesXY(ipMover[nMoverIndex].std.P_SetPosition.x,fTileLengthY*(nZoneRow-nZoneCounter)/nZoneRow-(nSizeOfMover+1)/2-1);
		ipMover[nMoverIndex].std.MoveToPosition('',
																	pos,
																	InitVelo,
																	InitAcc,
																	InitAcc,
																	InitJerk);
		nCounterX[nZoneCounter+1]:=nCounterX[nZoneCounter+1]+1;
		nMoverIistInZone[k]:=nMoverIndex;
		k:=k+1;
		SortingState:=50;
	
	50:
		IF 	ipMover[nMoverIndex].std.P_MoveToPosition.Done THEN 
			SortingState:=20;	
		END_IF


///////////////////////************sorting movers in every zone*************/////////////////////////////				
	60:
		fbMoverSortList[nZoneCounter+1]:=M_SortingInZone(nCounterX[nZoneCounter+1],nMoverIistInZone,ipMover);
		FOR i := 1 TO nCounterX[nZoneCounter+1] DO
				fbMoverSortList[nZoneCounter+1].M_AddToList(fbMoverSortList[nZoneCounter+1].List[i]);
		END_FOR
		k:=1;
		nZoneCounter:=nZoneCounter+1;
		IF nZoneRow - nZoneCounter > 0 THEN
			nMoverIndex:=0;			
			SortingState:=20;
			ELSE
			nZoneCounter:=0;
			SortingState:=110;				
		END_IF


///////////////////////************Movers move to left of the zone in turn*************/////////////////////////////				
	110:
		IF InitList.List[0]>0 THEN 
			SortingState:=120;
		END_IF
		
	120:
		nZoneCounter:=nZoneCounter+1;
		IF nZoneRow - nZoneCounter >= 0 THEN	
			SortingState:=130;
			ELSE
			SortingState:=200;	
		END_IF		

	130:
		IF nCounterX[nZoneCounter] = 0 THEN
					SortingState:=120;				
			ELSE
				FOR i:=1 TO nCounterX[nZoneCounter] DO
					Pos.SetValuesXY((i-1)*fTileLengthX/INT_TO_LREAL(nZoneColumn)+(fTileLengthX/INT_TO_LREAL(nZoneColumn)+1)/2+2,ipMover[fbMoverSortList[nZoneCounter].List[i]].std.P_SetPosition.y);
					ipMover[fbMoverSortList[nZoneCounter].List[i]].std.MoveToPosition('',
																				pos,
																				InitVelo,
																				InitAcc,
																				InitAcc,
																				InitJerk);
					SortingState:=150;		
				END_FOR				
		END_IF


	150:
		bDone:=TRUE;
		FOR i:=1 TO nCounterX[nZoneCounter] DO
			bDone := bDone AND ipMover[fbMoverSortList[nZoneCounter].List[i]].std.P_MoveToPosition.Done;
		END_FOR
		IF bDone THEN
			SortingState:=120;
		END_IF
		

///////////////////////************Movers move to table point in turn*************/////////////////////////////		
	200:
//		FOR i := 1 TO  nZoneRow DO
//			IF nCounterX[i]- nSorting[i] > 0 THEN
//				bGive:=TRUE;
//				nGive:=i;
//			ELSIF	nCounterX[i]- nSorting[i] < 0 THEN
//				bGet:=TRUE;		
//				nGet:=i;
//			ELSE
//				;
//			END_IF
//			IF bGive AND bGet THEN
//				bGive:=FALSE;
//				bGet:=FALSE;
//				SortingState:=210;
//				EXIT;
//			END_IF
//		END_FOR
		FOR i := 1 TO  nZoneRow DO
			IF nCounterX[i]- nSorting[i] > 0 THEN
				bGive:=TRUE;
				bFirstGive := TRUE;
				nGive:=i;
				EXIT;
			ELSIF	nCounterX[i]- nSorting[i] < 0 THEN
				bGet:=TRUE;	
				bFirstGet := TRUE;	
				nGet:=i;
				EXIT;
			ELSE
				;
			END_IF
		END_FOR

		FOR j := i TO  nZoneRow DO
			IF bFirstGive AND nCounterX[j]- nSorting[j] < 0 THEN
				bGet:=TRUE;		
				nGet:=j;		
			END_IF		
			IF bFirstGet AND nCounterX[j]- nSorting[j] > 0 THEN
				bGive:=TRUE;
				nGive:=j;		
			END_IF		
		END_FOR
		
		IF bGive AND bGet THEN
			bGive:=FALSE;
			bGet:=FALSE;
			SortingState:=210;
		END_IF
		
		IF MEMCMP(ADR(nCounterX) , ADR(nSorting),SIZEOF(nSorting)) = 0 THEN	
				SortingState:=500;					
		END_IF		
		
	210:
		IF nGive > nGet THEN
				nMAXTemp := nCounterX[nGet];
				nMAX := nGet; 				
				FOR i := nGet TO nGive BY 1 DO
					IF i + 1 <= nGive THEN
						IF nMAXTemp <= nCounterX[i+1] THEN
							nMAXTemp := nCounterX[i+1];
							nMAX := i + 1;
//							ELSE
//							nMAX := i; 	
						END_IF	
					END_IF
				END_FOR	
//		nPos:=nCounterX[nMAX] - nCounterX[nGet]+1;
//		IF nMAX - nGet = 0 THEN
//			nPos := 0;
//		END_IF				
			ELSE
					nMAXTemp := nCounterX[nGive];
					nMAX := nGive; 
				FOR i := nGive TO nGet BY 1 DO
					IF i + 1 <= nGet THEN
						IF nMAXTemp <= nCounterX[i+1] THEN
							nMAXTemp := nCounterX[i+1];
							nMAX := i + 1;
//							ELSE
//							nMAX := i; 								
						END_IF	
					END_IF
				END_FOR	

						
		END_IF
		
		nPos:=nCounterX[nMAX] - nCounterX[nGive]+1;
		IF nMAX = nGive AND NOT (nCounterX[nGive] = nCounterX[nGet]) THEN		
				nPos := 0;			
		END_IF
//		nPos:=nCounterX[nMAX] - nCounterX[nGive]+1;
//		IF nCounterX[nMAX] - nCounterX[nGive] = 0 THEN
//			nPos := 0;
//		END_IF
		nMoverIndex:=fbMoverSortList[nGive].List[nCounterX[nGive]];
		fLengthGive:=ipMover[nMoverIndex].std.P_SetPosition.x+nPos*fTileLengthX/INT_TO_LREAL(nZoneColumn)+7;
		fLengthY:=ipMover[nMoverIndex].std.P_SetPosition.y;
		Pos.SetValuesXY(fLengthGive,fLengthY);
		SortingState:=220;		
	
	220:
		ipMover[nMoverIndex].std.MoveToPosition('',
																	Pos,
																	InitVelo,
																	InitAcc,
																	InitAcc,
																	InitJerk);	

		SortingState:=221;
		
	221:
		IF 	ipMover[nMoverIndex].std.P_MoveToPosition.Done THEN 
			SortingState:=230;	
		END_IF
		
	230:
		fLengthY:=ipMover[nMoverIndex].std.P_SetPosition.y+INT_TO_LREAL(nGive-nGet)*fTileLengthY/INT_TO_LREAL(nZoneRow);					
		Pos.SetValuesXY(ipMover[nMoverIndex].std.P_SetPosition.x,fLengthY);
//		Pos.SetValuesXY(fLengthGive,fLengthY);		
		SortingState:=240;		
		
		
	240:
		ipMover[nMoverIndex].std.MoveToPosition('',
																	Pos,
																	InitVelo,
																	InitAcc,
																	InitAcc,
																	InitJerk);	
		SortingState:=241;
		
	241:
		IF 	ipMover[nMoverIndex].std.P_MoveToPosition.Done THEN 
			SortingState:=250;	
		END_IF

	250:
		nPos:=ABS(nCounterX[nMAX] - nCounterX[nGet]);	
	
		IF nMAX = nGive THEN
			nPos:=ABS(nCounterX[nMAX] - nCounterX[nGet])-1;			
		END_IF

//		IF nGet > nGive AND nMAX = nGive THEN		
//			nPos:=ABS(nCounterX[nMAX] - nCounterX[nGet]);		
//		END_IF		
		
		IF nMAX = nGet  THEN
			nPos:=0;
		END_IF		
		fLengthGet:=ipMover[nMoverIndex].std.P_SetPosition.x-INT_TO_LREAL(nPos)*fTileLengthX/INT_TO_LREAL(nZoneColumn)-7;
		fLengthY:=ipMover[nMoverIndex].std.P_SetPosition.y;
		Pos.SetValuesXY(fLengthGet,fLengthY);
		SortingState:=260;		
		
	260:
		ipMover[nMoverIndex].std.MoveToPosition('',
																	Pos,
																	InitVelo,
																	InitAcc,
																	InitAcc,
																	InitJerk);			
				nCounterX[nGet]:=nCounterX[nGet]+1;
				nCounterX[nGive]:=nCounterX[nGive]-1;

//				fbMoverSortList[nGet].List[nCounterX[nGet]]:= nMoverIndex;
				nMoverIndex:=fbMoverSortList[nGive].M_RemoveLastFromList();
				fbMoverSortList[nGet].M_AddToList(nMoverIndex);	
				SortingState:=261;		

	261:
		IF 	ipMover[nMoverIndex].std.P_MoveToPosition.Done THEN 
			nGive := 0;
			nGet := 0;
			SortingState:=200;	
		END_IF	


	500:			
		M_MoverSorting:=TRUE;
END_CASE
END_METHOD

METHOD M_MoveToInitialPos : BOOL
VAR_INPUT
	
END_VAR
VAR_IN_OUT
	aManualPos							: ARRAY [*,*] OF REAL;
END_VAR
VAR_INST
	i,j,k							:INT;
	
	InitVelo							:LREAL;
	InitAcc,InitDec				:LREAL;
	InitJerk							:LREAL;
	
	PosArr								:PositionXYC;
	IsAllArrived					: BOOL;
END_VAR
	InitVelo:=SetInitVelo;
	InitAcc:=SetInitAccDec;
	InitDec:=SetInitAccDec;
	InitJerk:=SetInitJerk;

CASE MovingState OF
	0:
		i := i + 1;
		IF nCounterX[i]<> 0 THEN			
			k := k + nCounterX[i];
			FOR j := 1 TO nCounterX[i] DO
				PosArr.SetValuesXY(aManualPos[k+1-j,1],aManualPos[k+1-j,2]);	
				ipMover[fbMoverSortList[i].List[nCounterX[i]+1-j]].std.MoveToPosition('',
								PosArr,
								InitVelo,
								InitAcc,
								InitAcc,
								InitJerk);					
			END_FOR
		END_IF
		MovingState:=10;
	
	10:
		IF i > nZoneRow THEN
				MovingState:=20;	
			ELSE
				MovingState:=0;	
		END_IF	
		
	20:
		k := 0;
		i := 0;		
		IsAllArrived:=TRUE;
			FOR j:=1 TO TO_INT(Tc3_XPlanarStandard.Params_XPlanar.moverCount) DO 	
				IsAllArrived:=IsAllArrived AND ipMover[j].std.P_MoveToPosition.Done;
			END_FOR	

		IF IsAllArrived THEN 
				MovingState:=50;								
		END_IF


	50:
		M_MoveToInitialPos := TRUE;
		
	
	
	
END_CASE
END_METHOD

METHOD M_SortingInZone : FB_MoverList
VAR_INPUT
	nNumber													: INT;
	nMoverList													: ARRAY[0..MAX_MOVERS] OF INT;
	ipMover														: ARRAY [0..MAX_MOVERS] OF I_XPlanarMover;		
END_VAR
VAR
	MoverList													: ARRAY[0..MAX_MOVERS] OF INT;
	MoverListMem												: ARRAY[0..MAX_MOVERS] OF INT;
	IdMem															: INT;
	i,j,K,L,M,N														: INT;
END_VAR
MEMSET(ADR(MoverList),0,SIZEOF(MoverList));
MEMCPY(ADR(MoverList),ADR(nMoverList),SIZEOF(nMoverList));
//FOR  M:=1 TO nNumber DO 
//		MoverList[0]										:=MoverList[0]+1;
//		MoverList[MoverList[0]]											:=M;
//END_FOR


FOR i:=1 TO nNumber-1 DO 
	FOR j := 1 TO nNumber-i DO
		IF ipMover[MoverList[j]].std.P_SetPosition.x>ipMover[MoverList[j+1]].std.P_SetPosition.x THEN 
			IdMem							:=MoverList[j];
			MoverList[j]					:=MoverList[j+1];
			MoverList[j+1]				:=IdMem;
		END_IF
	END_FOR
END_FOR	




//IF NOT EnableBackwards THEN 
	MoverListMem[0]							:=MoverList[0];
	FOR L:=1 TO nNumber  DO 
		MoverListMem[L]						:=MoverList[l];
	END_FOR
//ELSE
//	MEMCPY(ADR(MoverListMem[1]),ADR(MoverList[MAX_MOVERS_NUMBER- MoverList[0] +1]),SIZEOF(MoverListMem[1])*MoverList[0]);
//	MoverListMem[0]							:=MoverList[0];
//END_IF

M_SortingInZone.M_CopyList(MoverListMem);
END_METHOD

END_FUNCTION_BLOCK

// ---- Logic/Initialize/FB_MoverList.TcPOU
FUNCTION_BLOCK FB_MoverList
VAR_OUTPUT	
	List									: ARRAY[0..MAX_MOVERS] OF INT; //starts from 0, element zero is the number in the list 
END_VAR
VAR
	i: INT;
END_VAR

// Adding and removing stuff to a list can be a difficult as such a block has 
// been built with methods to add/remove from a list. 
// list acts like a FIFO, the list is filled from the back and emptied from the front.

METHOD M_AddToList
VAR_INPUT
	IDToAdd: INT;
END_VAR
// Movers are handled in a FIFO manner new movers are added to the end of the list 
List[0] 					:= List[0] +1; //List[0] holds the number of movers in the list 
List[List[0]] 				:= IDToAdd; //whern there is 1 in the list, List[0] = 1 and LIst[1] = IDToAdd
END_METHOD

METHOD M_ClearList
MEMSET(destAddr:=ADR(List),fillByte:=0,n:=SIZEOF(List));
END_METHOD

METHOD M_CopyList
VAR_INPUT
	ListToCopy: ARRAY[0..MAX_MOVERS] OF INT;
END_VAR
// method to copy a complete list, don't allow an extrnal copy unless its with a method
List := ListToCopy;
END_METHOD

METHOD M_GetFirstInList : INT
M_GetFirstInList := List[1];
END_METHOD

METHOD M_RecycleDown : BOOL
VAR
	iTemp: INT;
END_VAR
iTemp							:= List[MAX_MOVERS];
MEMCPY(ADR(List[2]),ADR(List[1]),SIZEOF(List)-SIZEOF(List[1])*2);
List[1]							:=iTemp;
M_RecycleDown					:= TRUE;
END_METHOD

METHOD M_RemoveFromList : INT
VAR
	I: INT;
END_VAR
//If there is something in the list, get the first element 
IF List[0] >= 1 THEN 
	M_RemoveFromList := List[1]; //List [1] is the first in the list, list[0] contains the number of items in the list  
	MEMCPY(ADR(List[1]),ADR(List[2]),SIZEOF(List)- 2 * SIZEOF(List[1])); //start at address 2 and copy the size of the list minus elements 0 and 1 
	List[MAX_MOVERS] := -1; //the last item in the list is now -1 
	List[0] := List[0]-1; // there is now one less item in the list 
ELSE //there was nothing in the list, return an invalid mover number 
	M_RemoveFromList := -1;// return an invalid mover 
END_IF
END_METHOD

METHOD M_RemoveLastFromList : int
VAR_INPUT
END_VAR
IF List[0] >= 1 THEN 
	M_RemoveLastFromList := List[ List[0]]; //List [1] is the first in the list, list[0] contains the number of items in the list  
	List[ List[0]]:=0;
	List[0]:=List[0]-1;
ELSE //there was nothing in the list, return an invalid mover number 
	M_RemoveLastFromList := -1;// return an invalid mover 
END_IF
END_METHOD

METHOD M_ReverseList : BOOL
VAR
	TempList: ARRAY[0..MAX_MOVERS] OF INT;
END_VAR
 
TempList:=List;
FOR i:=1 TO TempList[0] DO
	List[i]						:=TempList[TempList[0]+1-i];
END_FOR
M_ReverseList					:= TRUE;
END_METHOD

PROPERTY P_NumInList : INT
GET
P_NumInList:= List[0];
END_GET
END_PROPERTY

END_FUNCTION_BLOCK

// ---- Machine/EquipmentModules/CustomStations/FB_DecisionStation.TcPOU
FUNCTION_BLOCK FB_DecisionStation EXTENDS FB_XPlanarStationBase
VAR_INPUT
END_VAR
VAR_OUTPUT
END_VAR
VAR
	_OutputA	: I_XplanarStation;
	_OutputB	: I_XPlanarStation;
END_VAR

METHOD Execute
SUPER^.Execute(); //Call the base station logic to handle sending and receiving of movers

//When the station is in the Process mover state you can perform any application specific station logic
IF StationState = E_XPlanarStationState.ProcessMover THEN	
	IF ipCurrentMover.MoverIndex = 1 THEN			 
		ipNextStation := _OutputA;
	ELSE
		ipNextStation := _OutputB;
	END_IF
_StationComplete := TRUE;	//Set _StationComplete TRUE when done.  This will be automatically reset when the mover exits
END_IF
END_METHOD

PROPERTY OutputA : I_XPlanarStation
SET
_OutputA := OutputA;
END_SET
END_PROPERTY

PROPERTY OutputB : I_XPlanarStation
SET
_OutputB := OutputB;
END_SET
END_PROPERTY

END_FUNCTION_BLOCK

// ---- Machine/EquipmentModules/CustomStations/FB_SpinStation.TcPOU
FUNCTION_BLOCK FB_SpinStation EXTENDS FB_XPlanarStationBase
VAR_INPUT
END_VAR
VAR_OUTPUT
END_VAR
VAR
END_VAR

METHOD Execute
SUPER^.Execute();  //Call the base station logic to handle sending and receiving of movers

//When the station is in the Process mover state you can perform any application specific station logic
IF StationState = E_XPlanarStationState.ProcessMover THEN
	IF ipCurrentMover.Spin(NumOfTurns := 2) THEN
		_StationComplete := TRUE;  //Set _StationComplete TRUE when done.  This will be automatically reset when the mover exits
	END_IF
END_IF
END_METHOD

END_FUNCTION_BLOCK

// ---- Machine/EquipmentModules/FB_XPlanar_EM.TcPOU
FUNCTION_BLOCK FB_XPlanar_EM EXTENDS FB_PackML_BaseModule
VAR
    // Sub module definitions here

    // List of sub modules
    ipSubModules_Init : ARRAY[1..Parameters_PackML_Base.MAX_NO_OF_SUBMODULES] OF I_PackML_BaseModule := [];

    // Component definitions here
    XPlanarTable : FB_Component_Xplanar := (Name := 'XPlanarTable');
	
	//Station Components
	Station1	 : FB_DecisionStation	 := (Name := 'DecisionPoint');   //Declaration of a custom station
	Station2	 : FB_SpinStation 		 := (Name := 'RotateStation');
	Station3	 : FB_XPlanarStationBase := (Name := 'InspectStation');  //If no custom processing is needed simply declare an instance of the Station Base fb	 

    // List of Components
    ipComponents_Init : ARRAY[1..Parameters_PackML_Base.MAX_NO_OF_COMPONENTS] OF I_ComponentBase := [XPlanarTable, Station1, Station2, Station3];

    //Helper Vars
	Movers			  : ARRAY[1..Tc3_XPlanarStandard.Params_XPlanar.moverCount] OF FB_XPlanarMover;
	Tracks			  : ARRAY[1..Tc3_XPlanarStandard.Params_XPlanar.maxTrackCount] OF FB_XPlanarTrackSegment;
	
	
	fbinitbasic						: FB_BasicInitialization;
	aLocationOfArea 			: ARRAY[1..4,1..2] OF REAL:=[0,480,960,480,0,0,960,0];
	aManualPos					: ARRAY [1..19,1..2] OF REAL:=[60,420,240,420,420,420,600,420,860,420,60,300,240,300,420,300,600,300,860,300,60,180,240,180,420,180,600,180,860,180, 60,60,310,60,560,60,820,60];	
	
END_VAR

//! @summary This method contains code which will execute when this PackML module is in the <b>Aborting</b> state
METHOD PROTECTED Aborting
VAR
    i               : UDINT;
    SubModulesReady : BOOL := TRUE;
END_VAR

(*! <description> <b>Note:</b> The <i>Abort</i> command should be associated with the fault handing routine of a module. It should not be directly commanded from any user inteface. 

<table> 
	<tr>
		<th> Previous State </th>
		<th> Transition In </th>
		<th> Transition Out </th>
		<th> Next State  </th> 
	</tr>
	<tr>
		<td> <b>ANY</b> </td>
		<td> Abort Command </td> 
		<td> State Complete </td>
		<td> Aborted </td> 
	</tr>
</table>

This method is called as required by <c>StateControl()</c>
</description> 

*)
CASE DescendantSequenceState OF
    0:
        NoStateTasksToComplete  := FALSE;
        DescendantSequenceState := NextStep(DescendantSequenceState);

    10:
        IF XPlanarTable.Abort() THEN
            StateTasksComplete      := TRUE;
            DescendantSequenceState := NextStep(DescendantSequenceState);
        END_IF

    20:
        StateTasksComplete := TRUE;
END_CASE

SUPER^.Aborting();
END_METHOD

//! @summary This method contains code which will execute when this PackML module is in the <b>Clearing</b> state
METHOD PROTECTED Clearing
VAR
    i               : UDINT;
    SubModulesReady : BOOL := TRUE;
END_VAR

(*! <description> <b>Note:</b> The <i>Clear</i> command can also be thought of as a <i>fault reset</i> depite the ambiguity in the naming of the <i>Reset</i> state. 
<table> 
	<tr>
		<th> Previous State </th>
		<th> Transition In </th>
		<th> Transition Out </th>
		<th> Next State  </th> 
	</tr>
	<tr>
		<td> Aborted </td>
		<td> Clear Command </td> 
		<td> State Complete </td>
		<td> Stopped </td> 
	</tr>
</table>
This method is called as required by <c>StateControl()</c>
</description> 

*)
CASE _CurrentMode OF
    E_PMLUnitMode.ePMLUnitMode_Production:
        CASE DescendantSequenceState OF
            0: //Init
                NoStateTasksToComplete  := FALSE;
                XPlanarTable._Error     := FALSE;
				Station1.Reset();
				Station2.Reset();
				Station3.Reset();
			
                DescendantSequenceState := NextStep(DescendantSequenceState);

            10: //Check for Track initialization
                IF NOT XPlanarTable.TracksInitialized THEN
                    DescendantSequenceState := NextMinorStep(DescendantSequenceState);
                ELSE
                    DescendantSequenceState := NextStep(DescendantSequenceState);
                END_IF

            11: //Build Track Segments
                IF XPlanarTable.BuildTracks() THEN
                    IF NOT XPlanarTable.Error THEN
                      DescendantSequenceState := NextStep(DescendantSequenceState);
                    ELSE
                        DescendantSequenceState := 999;
                    END_IF;
                END_IF

            20: //Enable Group
                IF XPlanarTable.EnableGroup() THEN
                    DescendantSequenceState := NextStep(DescendantSequenceState);
                END_IF

            30:
                //Clearing complete
				fbinitbasic(bReset:=TRUE);
                StateTasksComplete := TRUE;
        END_CASE

    E_PMLUnitMode.ePMLUnitMode_Manual:
        ;
END_CASE

SUPER^.Clearing();
END_METHOD

METHOD PROTECTED CreateEvents
VAR_INPUT
END_VAR
// Add your event creation here

// Super call to base
SUPER^.CreateEvents();
END_METHOD

METHOD CyclicLogic
VAR
    i : INT;
    j : UDINT;
END_VAR
IF NOT _InitComplete THEN
    _InitComplete := Initialize();
END_IF

SUPER^.CyclicLogic();

IF _InitComplete THEN
	FOR j := 1 TO MAX_STATION_NUMBER DO
		stStationVis[j].bInit := TRUE;
		stStationVis[j].fPosition_X := stStationPos[j].fpositionX;		
		stStationVis[j].fPosition_Y := stStationPos[j].fpositionY;		
	END_FOR
	FOR j := 1 TO Tc3_XPlanarStandard.Params_XPlanar.moverCount DO
		stMoverVis[j].fPosition_X := Movers[j].std.P_ActPosition.x;		
		stMoverVis[j].fPosition_Y := Movers[j].std.P_ActPosition.y;	
		stMoverVis[j].fPosition_C := Movers[j].std.P_ActPosition.c;			
	END_FOR	
	

END_IF
END_METHOD

//! @summary This method contains code which will execute when this PackML module is in the <b>Execute</b> state
METHOD PROTECTED Execute
VAR
    i : UDINT;
END_VAR
VAR_INST
	InspectSimTimer: TON;
END_VAR
(*! <description> <b>The base implementation of this method is empty. User must override this method to provide functionality.</b>
<table> 
	<tr>
		<th> Previous State </th>
		<th> Transition In </th>
		<th> Transition Out </th>
		<th> Next State  </th> 
	</tr>
	<tr>
		<td> Starting<b>-or-</b>Unholding <b>-or-</b>Unsuspending</td>
		<td> State Complete<i>(Starting<b>-or-</b>Unholding<b>-or-</b>Unsuspending)</i></td> 
		<td> State Complete<b>-or-</b>Hold Command<b>-or-</b>Suspend Command</td>
		<td> Completing<b>-or-</b>Holding<b>-or-</b>Suspending</td>
	</tr>
</table>
This method is called as required by <c>StateControl()</c>
</description> 

*)
CASE _CurrentMode OF
    E_PMLUnitMode.ePMLUnitMode_Production:
        FOR i := 1 TO Params_XPlanar.maxNumStation DO
            ip.Stations[i].Execute();
        END_FOR
	
	//Simulate the "Inspection Done" signal
	InspectSimTimer(IN := ip.Stations[3].StationReady, PT := T#1S);
	ip.Stations[3].StationComplete := InspectSimTimer.Q;
	
    E_PMLUnitMode.ePMLUnitMode_Manual:
        ;
END_CASE
END_METHOD

//! @summary Automatically enables and disables HMI control based on the PackML mode
METHOD PROTECTED HMIPermissions

//! @description This method is called cyclically by <c>CyclicLogic()</c>
//General Mode Based Monitoring and handling of HMI control
CASE _CurrentMode OF
    E_PMLUnitMode.ePMLUnitMode_Production:
        AllowHMIControl(ThisModuleOnly := FALSE);

    E_PMLUnitMode.ePMLUnitMode_Manual:
        AllowHMIControl(ThisModuleOnly := FALSE);

    E_PMLUnitMode.ePMLUnitMode_Maintenance:
        AllowHMIControl(ThisModuleOnly := FALSE);
END_CASE
END_METHOD

//! @summary Basic module initialization logic
METHOD PROTECTED Initialize : BOOL;
VAR
    i                        : UDINT;
    varInfo                  : __SYSTEM.VAR_INFO;
    AllSubUnitsInitialized   : BOOL := TRUE;
    AllComponentsInitialized : BOOL := TRUE;
    tmpMoveDynamics          : ST_MoveDynamics;
    stHaltDynamics           : ST_HaltDynamics;
END_VAR

//! @description This method is called by <c>CyclicLogic()</c> as required
Initialize := FALSE;
CASE DescendantSequenceState OF
	0:
		// Define the interfaces to the different subunits (Must take place before SUPER^.initialize call)
		FOR i := 1 TO SPT_BaseTypes.Parameters_PackML_Base.MAX_NO_OF_SUBMODULES DO
			ipSubModules[i] := ipSubModules_Init[i];
		END_FOR

		FOR i := 1 TO SPT_BaseTypes.Parameters_PackML_Base.MAX_NO_OF_COMPONENTS DO
			ipComponents[i] := ipComponents_Init[i];
		END_FOR

		_LogModeChanges			:= FALSE;
		_LogStateChanges		:= FALSE;
		DescendantSequenceState := DescendantSequenceState + 10;

	10:
		//Set Mover and Track interfaces
		FOR i := 1 TO Tc3_XPlanarStandard.Params_XPlanar.moverCount DO
			Movers[i].MoverIndex := i;
			ip.Movers[i]		  := Movers[i];
		END_FOR

		FOR i := 1 TO Tc3_XPlanarStandard.Params_XPlanar.maxTrackCount DO
			ip.Tracks[i] := Tracks[i];
		END_FOR

		DescendantSequenceState := DescendantSequenceState + 10;

	20:
		//Copy Mode names
		FOR i := 1 TO 3 DO
			ModeNames[i] := F_UnitModeToString(UDINT_TO_DINT(i));
		END_FOR

		DescendantSequenceState := DescendantSequenceState + 10;

	30:
		//Call the Super
		IF SUPER^.Initialize() THEN
			DescendantSequenceState := DescendantSequenceState + 10;
		END_IF

	40:
		IF SetupTrackSegments() THEN
			DescendantSequenceState := DescendantSequenceState + 10;
		END_IF

	50:
		IF SetupStations() THEN
			DescendantSequenceState := DescendantSequenceState + 10;
		END_IF

	60:
		stHaltDynamics.PathXY.fVelocity		:= 500.0;
		stHaltDynamics.PathXY.fAcceleration := 10000.0;
		stHaltDynamics.PathXY.fDeceleration := 10000.0;
		stHaltDynamics.PathXY.fJerk			:= 100000.0;
		stHaltDynamics.AxisX.fVelocity		:= 500.0;
		stHaltDynamics.AxisX.fAcceleration	:= 10000.0;
		stHaltDynamics.AxisX.fDeceleration	:= 10000.0;
		stHaltDynamics.AxisX.fJerk			:= 100000.0;
		stHaltDynamics.AxisY.fVelocity		:= 500.0;
		stHaltDynamics.AxisY.fAcceleration	:= 10000.0;
		stHaltDynamics.AxisY.fDeceleration	:= 10000.0;
		stHaltDynamics.AxisY.fJerk			:= 100000.0;
		stHaltDynamics.AxisZ.fVelocity		:= 500.0;
		stHaltDynamics.AxisZ.fAcceleration	:= 10000.0;
		stHaltDynamics.AxisZ.fDeceleration	:= 10000.0;
		stHaltDynamics.AxisZ.fJerk			:= 100000.0;
		stHaltDynamics.AxisA.fVelocity		:= 10.0;
		stHaltDynamics.AxisA.fAcceleration	:= 100.0;
		stHaltDynamics.AxisA.fDeceleration	:= 100.0;
		stHaltDynamics.AxisA.fJerk			:= 100.0;
		stHaltDynamics.AxisB.fVelocity		:= 10.0;
		stHaltDynamics.AxisB.fAcceleration	:= 100.0;
		stHaltDynamics.AxisB.fDeceleration	:= 100.0;
		stHaltDynamics.AxisB.fJerk			:= 100.0;
		stHaltDynamics.AxisC.fVelocity		:= 36.0;
		stHaltDynamics.AxisC.fAcceleration	:= 360.0;
		stHaltDynamics.AxisC.fDeceleration	:= 360.0;
		stHaltDynamics.AxisC.fJerk			:= 360.0;
		FOR i := 1 TO Params_XPlanar.moverCount DO
			ip.Movers[i].std.P_HaltDynamics := stHaltDynamics;
		END_FOR

		Initialize := TRUE;
END_CASE
END_METHOD

//! @summary This method contains code which will execute when this PackML module is in the <b>Resetting</b> state
METHOD PROTECTED Resetting
VAR
	SubModulesReady : BOOL := TRUE;
END_VAR

VAR_INST
	i : UDINT;
END_VAR

(*! <description> <b>Note:</b> The <i>Reset</i> command can also be thought of as an <i>enable</i> depite the ambiguity in the naming of the <i>Clearing</i> state.
<table> 
	<tr>
		<th> Previous State </th>
		<th> Transition In </th>
		<th> Transition Out </th>
		<th> Next State  </th> 
	</tr>
	<tr>
		<td> Stopped<b>-or-</b>Completed </td>
		<td> Reset Command </td> 
		<td> State Complete </td>
		<td> Idle </td> 
	</tr>
</table>
This method is called as required by <c>StateControl()</c>
</description> 

*)
CASE _CurrentMode OF
	E_PMLUnitMode.ePMLUnitMode_Production:
		CASE DescendantSequenceState OF
			0: //Init
				i						:= 1;
				NoStateTasksToComplete	:= FALSE;
				DescendantSequenceState := NextStep(DescendantSequenceState);

			10: //Reset XPlanar System
				IF XPlanarTable.Reset() THEN
					DescendantSequenceState := NextStep(DescendantSequenceState);
				END_IF

			20: //Enable Tracks
				IF XplanarTable.EnableTracks(FALSE) THEN
					DescendantSequenceState := NextStep(DescendantSequenceState);
				END_IF

			30: //Enable Movers
				IF XPlanarTable.EnableMovers(FALSE) THEN
					DescendantSequenceState := NextStep(DescendantSequenceState);
				END_IF

			40: //Check Mover Angle
				IF i <= Params_XPlanar.moverCount THEN
					IF ip.Movers[1].SquareUp() THEN
						DescendantSequenceState := NextMinorStep(DescendantSequenceState);
					END_IF
				ELSE
					DescendantSequenceState := NextStep(DescendantSequenceState);
				END_IF
				
			41: //CheckMoverCount
				IF i <= Params_XPlanar.moverCount THEN
					i := i + 1;
					DescendantSequenceState := 40;
				ELSE
					DescendantSequenceState := NextStep(DescendantSequenceState);
				END_IF				

			50: //Clearing complete
				StateTasksComplete := TRUE;
		END_CASE
END_CASE

SUPER^.Resetting();
END_METHOD

METHOD PRIVATE SetupStations : BOOL
VAR_INPUT
END_VAR
stStationPos[1].fpositionX:=120;
stStationPos[1].fpositionY:=240;
stStationPos[2].fpositionX:=360;
stStationPos[2].fpositionY:=360;
stStationPos[3].fpositionX:=360;
stStationPos[3].fpositionY:=120;






//Set Required Process Station Initialization Parameters
Station1.Position.SetValuesXYC(stStationPos[1].fpositionX, stStationPos[1].fpositionY, 0);		 //Set the center of the station
Station1.TrackID	 := ip.Tracks[1];				 //Set the interface of the track segment the station resides on
Station1.StationType := E_StationType.DecisionPoint; //Change the type to Decision Point only if the station is acting as a divert and processing on the fly
Station1.OutputA	 := Station2;					 //Set any custom station parameters
Station1.OutputB	 := Station3;
ip.Stations[1]		 := Station1; 					 //Register the station with the interface array

Station2.Position.SetValuesXYC(stStationPos[2].fpositionX, stStationPos[2].fpositionY, 0);
Station2.Size.x		 := 120;						 //Changes the station size in the X plane
Station2.Size.y		 := 120; 						 //Changes the station size in the Y plane
Station2.TrackID	 := ip.Tracks[2];
Station2.NextStation := Station1; 					 //Set the interface for the next station of the mover
ip.Stations[2]		 := Station2;

Station3.Position.SetValuesXYC(stStationPos[3].fpositionX, stStationPos[3].fpositionY, 0);
Station3.Size.x		 := 120;
Station3.Size.y		 := 120;
Station3.TrackID	 := ip.Tracks[3];
Station3.NextStation := Station1;
ip.Stations[3]		 := Station3;
SetupStations		 := TRUE;
END_METHOD

METHOD PRIVATE SetupTrackSegments : BOOL
VAR_INST
    nSegmentIndex : UDINT;
END_VAR

VAR
    ResultAddPoint : INT;
END_VAR
SetupTrackSegments := FALSE;
CASE nSegmentIndex OF
	0: //Get ready
		nSegmentIndex := nSegmentIndex + 1;

	//********************************************************************************************************************************

	//Add states for each track segment in the system

	//********************************************************************************************************************************
	1:
		ip.Tracks[nSegmentIndex].ID := nSegmentIndex;
		IF ip.Tracks[nSegmentIndex].TrackTable.ClearTrackTable() THEN
			ResultAddPoint := ip.Tracks[nSegmentIndex].TrackTable.AddPoint(E_PointType.Line_Start,
																		   E_PointOption.none,
																		   300,//480.0,
																		   120,//20.0,
																		   0.0);

			ResultAddPoint := ip.Tracks[nSegmentIndex].TrackTable.AddPoint(E_PointType.Line_End,
																		   E_PointOption.none,
																		   130,//240.0,
																		   120,//120.0,
																		   0.0);

			ResultAddPoint := ip.Tracks[nSegmentIndex].TrackTable.AddPoint(E_PointType.Line_Start,
																		   E_PointOption.none,
																		   120,//20.0,
																		   130,//240.0,
																		   0.0);

			ResultAddPoint := ip.Tracks[nSegmentIndex].TrackTable.AddPoint(E_PointType.Line_End,
																		   E_PointOption.none,
																		   120,//120.0,
																		   240,//480.0,
																		   0.0);

//			ResultAddPoint := ip.Tracks[nSegmentIndex].TrackTable.AddPoint(E_PointType.Line_Start,
//																		   E_PointOption.none,
//																		   120,//240.0,
//																		   300,//600.0,
//																		   0.0);

//			ResultAddPoint := ip.Tracks[nSegmentIndex].TrackTable.AddPoint(E_PointType.Line_End,
//																		   E_PointOption.none,
//																		   240,//480.0,
//																		   300,//600.0,
//																		   0.0);

			ip.Tracks[nSegmentIndex].TrackTable.P_CloseTheLoop := FALSE;
		END_IF

		nSegmentIndex := nSegmentIndex + 1;

	2:
		ip.Tracks[2].ID := 2;  															//Set the ID property of the track segment
		IF ip.Tracks[2].TrackTable.ClearTrackTable() THEN								//Clean up any stray points in the table
			ResultAddPoint := ip.Tracks[2].TrackTable.AddPoint(E_PointType.Line_Start,	//Configure track points
															   E_PointOption.none,
															   120,//600.0,
															   240,//480.0,
															   0.0);

			ResultAddPoint := ip.Tracks[2].TrackTable.AddPoint(E_PointType.Line_End,
															   E_PointOption.none,
															   120,//600.0,
															   350,//240.0,
															   0.0);
															   
			ResultAddPoint := ip.Tracks[2].TrackTable.AddPoint(E_PointType.Line_Start,	//Configure track points
															   E_PointOption.none,
															   130,//600.0,
															   360,//480.0,
															   0.0);

			ResultAddPoint := ip.Tracks[2].TrackTable.AddPoint(E_PointType.Line_End,
															   E_PointOption.none,
															   360,//600.0,
															   360,//240.0,
															   0.0);			

			ResultAddPoint := ip.Tracks[2].TrackTable.AddPoint(E_PointType.Line_Start,	//Configure track points
															   E_PointOption.none,
															   360,//600.0,
															   330,//480.0,
															   0.0);

			ResultAddPoint := ip.Tracks[2].TrackTable.AddPoint(E_PointType.Line_End,
															   E_PointOption.none,
															   360,//600.0,
															   240,//240.0,
															   0.0);											   

			ip.Tracks[2].TrackTable.P_CloseTheLoop	 := FALSE;						//Set the segment close the loop property		
			ip.Tracks[2].TrackTable.P_StartFromTrack := ip.Tracks[1].std;			//If linking to a previous track segment set the interface
			ip.Tracks[2].TrackTable.P_EndAtTrack	 := ip.Tracks[1].std;			//If linking to a downstream track segment set the interface
		END_IF

		nSegmentIndex := nSegmentIndex + 1;

	3:
		ip.Tracks[nSegmentIndex].ID := nSegmentIndex;
		IF ip.Tracks[nSegmentIndex].TrackTable.ClearTrackTable() THEN
			ResultAddPoint := ip.Tracks[nSegmentIndex].TrackTable.AddPoint(E_PointType.Line_Start,
																		   E_PointOption.none,
																		   140,//480.0,
																		   240,//600.0,
																		   0.0);

			ResultAddPoint := ip.Tracks[nSegmentIndex].TrackTable.AddPoint(E_PointType.Line_End,
																		   E_PointOption.none,
																		   350,//720.0,
																		   240,//600.0,
																		   0.0);

			ResultAddPoint := ip.Tracks[nSegmentIndex].TrackTable.AddPoint(E_PointType.Line_Start,
																		   E_PointOption.none,
																		   360,//840.0,
																		   230,//480.0,
																		   0.0);

			ResultAddPoint := ip.Tracks[nSegmentIndex].TrackTable.AddPoint(E_PointType.Line_End,
																		   E_PointOption.none,
																		   360,//840.0,
																		   120,//240.0,
																		   0.0);

//			ResultAddPoint := ip.Tracks[nSegmentIndex].TrackTable.AddPoint(E_PointType.Line_Start,
//																		   E_PointOption.none,
//																		   360,//720.0,
//																		   60,//120.0,
//																		   0.0);

//			ResultAddPoint := ip.Tracks[nSegmentIndex].TrackTable.AddPoint(E_PointType.Line_End,
//																		   E_PointOption.none,
//																		  240,// 480.0,
//																		   60,//120.0,
//																		   0.0);

			ip.Tracks[nSegmentIndex].TrackTable.P_CloseTheLoop	 := FALSE;
			ip.Tracks[nSegmentIndex].TrackTable.P_StartFromTrack := ip.Tracks[1].std;
			ip.Tracks[nSegmentIndex].TrackTable.P_EndAtTrack	 := ip.Tracks[1].std;
		END_IF

		nSegmentIndex := nSegmentIndex + 1;
		
	4:
		ip.Tracks[nSegmentIndex].ID := nSegmentIndex;
		IF ip.Tracks[nSegmentIndex].TrackTable.ClearTrackTable() THEN
			ResultAddPoint := ip.Tracks[nSegmentIndex].TrackTable.AddPoint(E_PointType.Line_Start,
																		   E_PointOption.none,
																		   60,//100.0,
																		   420,//100.0,
																		   0.0);

			ResultAddPoint := ip.Tracks[nSegmentIndex].TrackTable.AddPoint(E_PointType.Line_End,
																		   E_PointOption.none,
																		   420,//100.0,
																		   420,//500.0,
																		   0.0);

			ResultAddPoint := ip.Tracks[nSegmentIndex].TrackTable.AddPoint(E_PointType.Line_Start,
																		   E_PointOption.none,
																		   420,//240.0,
																		   300,//620.0,
																		   0.0);

			ResultAddPoint := ip.Tracks[nSegmentIndex].TrackTable.AddPoint(E_PointType.Line_End,
																		   E_PointOption.none,
																		   60,//780.0,
																		   300,//620.0,
																		   0.0);

			ResultAddPoint := ip.Tracks[nSegmentIndex].TrackTable.AddPoint(E_PointType.Line_Start,
																		   E_PointOption.none,
																		   60,//860.0,
																		   180,//480.0,
																		   0.0);

			ResultAddPoint := ip.Tracks[nSegmentIndex].TrackTable.AddPoint(E_PointType.Line_End,
																		   E_PointOption.none,
																		   420,//860.0,
																		   180,//240.0,
																		   0.0);
																		   
			ResultAddPoint := ip.Tracks[nSegmentIndex].TrackTable.AddPoint(E_PointType.Line_Start,
																		   E_PointOption.none,
																		   420,//860.0,
																		   60,//240.0,
																		   0.0);					

			ResultAddPoint := ip.Tracks[nSegmentIndex].TrackTable.AddPoint(E_PointType.Line_End,
																		   E_PointOption.none,
																		   60,//860.0,
																		   60,//240.0,
																		   0.0);													

			ip.Tracks[nSegmentIndex].TrackTable.P_CloseTheLoop	 := FALSE;
			ip.Tracks[nSegmentIndex].TrackTable.P_EndAtTrack	 := ip.Tracks[1].std;
		END_IF

		nSegmentIndex := nSegmentIndex + 1;		

	5:
		nSegmentIndex	   := 0;
		SetupTrackSegments := TRUE;
END_CASE
END_METHOD

//! @summary This method contains code which will execute when this PackML module is in the <b>Starting</b> state
METHOD PROTECTED Starting
VAR
    SubModulesReady : BOOL := TRUE;
    Position        : PositionXYC;
    check           : ST_CheckStartConditionFeedback;
    lError          : BOOL;
    lErrorID        : UDINT;
    Angle           : LREAL;
END_VAR

VAR_INST
    MoverNumber       : UDINT;
    StationNumber     : UDINT;
    ipMover           : ARRAY [0..Tc3_XPlanarStandard.Params_XPlanar.moverCount] OF I_XPlanarMover;
    ipStation         : I_XPlanarStation;
    JoinState         : INT;
    MoveState         : INT;
    i                 : UDINT;
    JoinTrackNum      : UINT;
    MoveStationNum    : ARRAY[1..Params_XPlanar.moverCount] OF UINT;
    MoveStationNeeded : ARRAY[1..Params_XPlanar.moverCount] OF BOOL;
    JoinStationNeeded : ARRAY[1..Params_XPlanar.moverCount] OF BOOL;
END_VAR
CASE _CurrentMode OF
	E_PMLUnitMode.ePMLUnitMode_Production:
		CASE DescendantSequenceState OF
			0:
				NoStateTasksToComplete	:= FALSE;
				DescendantSequenceState := 10;
				StationNumber			:= 1;
				i						:= 1;
				JoinState				:= 0;

			10: //Clean Up Mover Queues
				FOR i := 1 TO Params_XPlanar.moverCount DO
					ip.Movers[i].Destination := 0;
				END_FOR

				FOR i := 1 TO Params_XPlanar.maxNumStation DO
					ip.Stations[i].MoverQueue.Dequeue();
				END_FOR

				i						:= 1;
				DescendantSequenceState := 15;
//				DescendantSequenceState := NextStep(DescendantSequenceState);
				
			15:
				fbinitbasic(bExcute:=TRUE,nSizeOfMover:=115,aLocationOfArea:=aLocationOfArea,ipMover:=ip.Movers,aManualPos:=aManualPos,bReset:=);
				IF fbinitbasic.Done THEN
//						DescendantSequenceState := NextStep(DescendantSequenceState);		
				END_IF
			

			20: //Join Movers to recovery track
				IF i <= Params_XPlanar.moverCount THEN
					IF ip.Movers[i].JoinTrack(ip.Tracks[4]) THEN
						DescendantSequenceState := NextMinorStep(DescendantSequenceState);
					END_IF
				ELSE
					i						:= 1;
					DescendantSequenceState := NextStep(DescendantSequenceState);
				END_IF
				
			21: //Check Mover Count
				IF i <= Params_XPlanar.moverCount THEN
 					i := i + 1;
					DescendantSequenceState := 20;
				ELSE
					i						:= 1;
					DescendantSequenceState := NextStep(DescendantSequenceState);
				END_IF					

			30: //Send Movers around to station 1
				IF i <= Params_XPlanar.moverCount THEN
					IF ip.Movers[i].SendToStation(ip.Stations[1]) THEN
						DescendantSequenceState := NextMinorStep(DescendantSequenceState);
					END_IF
				ELSE
					i						:= 1;
					DescendantSequenceState := NextStep(DescendantSequenceState);
				END_IF
				
			31: //Check Mover Count
				IF i <= Params_XPlanar.moverCount THEN
 					i := i + 1;
					DescendantSequenceState := 30;
				ELSE
					i						:= 1;
					DescendantSequenceState := NextStep(DescendantSequenceState);
				END_IF	

			40:
				StateTasksComplete := TRUE;
		END_CASE

	E_PMLUnitMode.ePMLUnitMode_Manual:
		;
END_CASE

SUPER^.Starting();
END_METHOD

END_FUNCTION_BLOCK

// ---- NextStep.TcPOU
FUNCTION NextStep : UDINT
VAR_INPUT
	StateVar	: UDINT;
END_VAR
VAR
END_VAR

NextStep := ((StateVar / 10)* 10) + 10;

END_FUNCTION

// ---- NextMinorStep.TcPOU
FUNCTION NextMinorStep : UDINT
VAR_INPUT
	StateVar	: UDINT;
END_VAR
VAR
END_VAR

NextMinorStep := StateVar + 1;

END_FUNCTION

// ---- Machine/FB_Machine.TcPOU
FUNCTION_BLOCK FB_Machine EXTENDS FB_PackML_BaseModule
VAR
    (*Sub Modules*)
    XPlanar : FB_XPlanar_EM := (Name := 'XPlaner EM');

    (*Initial List of SubModules*)

    //Add list of EMs here...
    ipSubModules_Init : ARRAY[1..Parameters_PackML_Base.MAX_NO_OF_SUBMODULES] OF I_PackML_BaseModule := [XPlanar];

    // Components

    //Add list of components here...
    ipComponents_Init : ARRAY[1..Parameters_PackML_Base.MAX_NO_OF_COMPONENTS] OF I_ComponentBase := [];

    // Local and Simulation variables

    (*Alarms for this module*)
    MachineAlarms : ARRAY[1..MACHINE_ALARM_COUNT] OF FB_TcAlarm;
    RecipeLoaded  : BOOL := FALSE;

    //Pack Tags for System
    {attribute 'OPC.UA.DA' := '1'}
    _PackTags : ST_PackMLv30Ext; //ST_PackMLv30 is obsolete in Tc3_PackML_V2
END_VAR

VAR CONSTANT
    //Alarm count constant
    MACHINE_ALARM_COUNT : INT := 1; //Change this value based on how many alarms are in your machine
END_VAR

METHOD PROTECTED CreateEvents
VAR_INPUT
END_VAR
// Add your event creation here
F_CreateAllEventsInClass(Alarms     := MachineAlarms,
                         ClassSize  := SIZEOF(TC_EVENTS.MachineAlarms),
                         pInitEvent := ADR(TC_EVENTS.MachineAlarms.InitReferenceEvent),
                         Prefix     := Name);

// Super call to base
SUPER^.CreateEvents();
END_METHOD

METHOD CyclicLogic
VAR
    NewSeverity    : TCEventSeverity;
    AlarmResponses : ARRAY[0..4] OF E_AlarmResponse; //Temporary response array	
END_VAR
IF NOT _InitComplete THEN
    _InitComplete := Initialize();
    RETURN;
END_IF

_CurrentAlarmSeverity := F_GetMaxSeverityRaised(MachineAlarms, NewSeverity);
SUPER^.CyclicLogic();
_PackTags.Status.StateCurrent    := _CurrentState;
_PackTags.Status.UnitModeCurrent := _CurrentMode;
UpdateModeTimers();
END_METHOD

METHOD PROTECTED HMIPermissions
VAR_INPUT
END_VAR
//General Mode Based Monitoring and handling of HMI control
CASE _CurrentMode OF
    E_PMLUnitMode.ePMLUnitMode_Production:
        CASE _CurrentState OF
            E_PMLState.ePMLState_Stopped:
                AllowHMIControl(ThisModuleOnly := TRUE); //Allow control for recovery
            E_PMLState.ePMLState_Idle:
                AllowHMIControl(ThisModuleOnly := TRUE); //Allow control for recovery
            E_PMLState.ePMLState_Suspended:
                BlockHMIControl();

            E_PMLState.ePMLState_Execute:
                BlockHMIControl();

            E_PMLState.ePMLState_Aborted:
                AllowHMIControl(ThisModuleOnly := TRUE); //Allow control for recovery
            E_PMLState.ePMLState_Held:
                AllowHMIControl(ThisModuleOnly := TRUE); //Allow control for recovery
            E_PMLState.ePMLState_Complete:
                BlockHMIControl();
        END_CASE

        AllowHMIControl(ThisModuleOnly := FALSE);

    E_PMLUnitMode.ePMLUnitMode_Manual:
        AllowHMIControl(ThisModuleOnly := FALSE);

    E_PMLUnitMode.ePMLUnitMode_Maintenance:
        AllowHMIControl(ThisModuleOnly := FALSE);
END_CASE
END_METHOD

METHOD PROTECTED Initialize : BOOL
VAR
    i : UDINT; //Generic iteration value
END_VAR
Initialize := FALSE;
CASE DescendantSequenceState OF
    0:
        // Define the interfaces to the different subunits (Must take place before SUPER^.initialize call)
        FOR i := 1 TO SPT_BaseTypes.Parameters_PackML_Base.MAX_NO_OF_SUBMODULES DO
            ipSubModules[i] := ipSubModules_Init[i];
        END_FOR

        FOR i := 1 TO SPT_BaseTypes.Parameters_PackML_Base.MAX_NO_OF_COMPONENTS DO
            ipComponents[i] := ipComponents_Init[i];
        END_FOR

        _LogModeChanges         := FALSE;
        _LogStateChanges        := FALSE;
        DescendantSequenceState := DescendantSequenceState + 10;

    10:
        //Setup Custom modes here
        DescendantSequenceState := DescendantSequenceState + 10;

    20:
        //Copy Mode names
        FOR i := 1 TO 3 DO
            ModeNames[i] := F_UnitModeToString(UDINT_TO_DINT(i));
        END_FOR

        DescendantSequenceState := DescendantSequenceState + 10;

    30:
        // Initialize Recipes 
        DescendantSequenceState := DescendantSequenceState + 10;

    40:
        //Call the Super
        IF SUPER^.Initialize() THEN
            DescendantSequenceState := DescendantSequenceState + 10;
        END_IF

    //Setup axes Master
    50:
        Initialize := TRUE;
END_CASE
END_METHOD

PROPERTY PUBLIC PackTags : ST_PackMLv30Ext
GET
PackTags := _PackTags;
END_GET
END_PROPERTY

//! @summary Provides fault reaction logic where the module state is driven to the <b>Stopping</b> state immediately
METHOD PROTECTED StopImmediate

//! @description No error is thrown by this fault reaction.

//! @description This method is called by <c>ComponentMonitor()</c> or <c>SubModuleMonitor()</c> as required
ChangeState(E_PMLCommand.ePMLCommand_Stop);
END_METHOD

METHOD PROTECTED SubModuleMonitor : BOOL
VAR
    AlarmResponses : ARRAY[0..4] OF E_AlarmResponse; //Temporary response array	
END_VAR

VAR
    Result : BOOL;
END_VAR
SubModuleMonitor := FALSE;

// Check the sub Modules for Alarm Severity
Result := SUPER^.SubModuleMonitor();

//Check the alarms at the machine level
_CurrentAlarmSeverity := F_GetMaxSeverityRaised(Alarms := MachineAlarms, CurrentSeverity := _CurrentAlarmSeverity);

//Check the severity of the machine level alarms
IF _CurrentState <> E_PMLState.ePMLState_Aborted AND _CurrentState <> E_PMLState.ePMLState_Aborting AND _CurrentState <> E_PMLState.ePMLState_Clearing AND
   _CurrentState <> E_PMLState.ePMLState_Stopped AND _CurrentState <> E_PMLState.ePMLState_Stopping THEN
    AlarmResponses := _ParentFaultResponseDefinitions;
    CASE AlarmResponses[CurrentAlarmSeverity] OF
        E_AlarmResponse.Abort_ImmediateError:
            AbortImmediateError(Name, TRUE);

        E_AlarmResponse.Abort_Immediate:
            AbortImmediate();

        E_AlarmResponse.Stop_Immediate:
            StopImmediate();

        E_AlarmResponse.Stop_Controlled:
            StopControlled();

        E_AlarmResponse.Hold_Immediate:
            HoldImmediate();

        E_AlarmResponse.Suspend_Immediate:
            SuspendImmediate();

        E_AlarmResponse.Suspend_Controlled:
            SuspendControlled();

        E_AlarmResponse.NoResponse:
            ;
    END_CASE
ELSIF _CurrentState = E_PMLState.ePMLState_Stopped OR _CurrentState = E_PMLState.ePMLState_Stopping THEN
    AlarmResponses := _ParentFaultResponseDefinitions;
    CASE AlarmResponses[CurrentAlarmSeverity] OF
        E_AlarmResponse.Abort_ImmediateError:
            AbortImmediateError(Name, TRUE);

        E_AlarmResponse.Abort_Immediate:
            AbortImmediate();

        E_AlarmResponse.NoResponse:
            ;
    END_CASE
END_IF
END_METHOD

METHOD UpdateModeTimers
VAR
    currentTime  : T_DCTIME64;
    timeToUpdate : LREAL;
END_VAR

VAR_INST
    lastTime  : T_DCTIME64 := F_GetActualDcTime64();
    lastState : DINT;
    lastMode  : DINT;
END_VAR

VAR
    Result : UDINT;
END_VAR
IF _PackTags.Status.StateCurrent <> lastState THEN
    Result    := MEMSET(ADR(_PackTags.Admin.StateCurrentTime), 0, SIZEOF(_PackTags.Admin.StateCurrentTime));
    lastState := _PackTags.Status.StateCurrent;
END_IF

IF _PackTags.Status.UnitModeCurrent <> lastMode THEN
    Result   := MEMSET(ADR(_PackTags.Admin.ModeCurrentTime), 0, SIZEOF(_PackTags.Admin.ModeCurrentTime));
    lastMode := _PackTags.Status.UnitModeCurrent;
END_IF

currentTime := F_GetActualDcTime64();
IF lastTime <> 0 THEN
    timeToUpdate := ULINT_TO_LREAL(currentTime - lastTime) / 1_000_000_000.0;
END_IF

// only seconds get added to the cumulative timers 
IF timeToUpdate > 1 THEN
    _PackTags.Admin.ModeCummulativeTime[_PackTags.Status.UnitModeCurrent] := _PackTags.Admin.ModeCummulativeTime[_PackTags.Status.UnitModeCurrent] + LREAL_TO_DINT(timeToUpdate);
    _PackTags.Admin.ModeCurrentTime[_PackTags.Status.UnitModeCurrent]     := _PackTags.Admin.ModeCurrentTime[_PackTags.Status.UnitModeCurrent] + LREAL_TO_DINT(timeToUpdate);
    _PackTags.Admin.StateCummulativeTime[_PackTags.Status.UnitModeCurrent, _PackTags.Status.StateCurrent]
        := _PackTags.Admin.StateCummulativeTime[_PackTags.Status.UnitModeCurrent, _PackTags.Status.StateCurrent] + LREAL_TO_DINT(timeToUpdate);

    _PackTags.Admin.StateCurrentTime[_PackTags.Status.UnitModeCurrent, _PackTags.Status.StateCurrent] :=
        _PackTags.Admin.StateCurrentTime[_PackTags.Status.UnitModeCurrent, _PackTags.Status.StateCurrent] + LREAL_TO_DINT(timeToUpdate);

    lastTime := currentTime;
END_IF
END_METHOD

END_FUNCTION_BLOCK

// ---- MAIN.TcPOU

PROGRAM MAIN
VAR
    // Machine Module
    Machine : FB_Machine := (Name := 'My First XPlanar Component Project');
    //Control Source for running machine
    ControlSourceHMI : FB_ControlSource;
    ControlSourcePB  : FB_ControlSource;
	
    //Local Vars
    InitComplete : BOOL;
END_VAR

{warning 'Simulation Demo Only - Lag monitoring is disabled'}

//All code runs from here.
CyclicLogic();

METHOD CyclicLogic
VAR_INPUT
END_VAR
IF NOT InitComplete THEN
    InitComplete := Initialize();
    RETURN;
END_IF

//Machine support HMI & Production Monitor
ControlSourcePB.CyclicLogic();
ControlSourceHMI.CyclicLogic();

//Machine Cyclic Logic
Machine.CyclicLogic();
END_METHOD

METHOD Initialize : BOOL
VAR_INPUT
END_VAR

VAR
    Result : BOOL;
END_VAR
//Top level machine initialization should happen here, in the main initialization METHOD. Each subsequent "layer" OF modules will be named within their respective "parent" intialize METHOD
IF NOT ControlSourceHMI.Registered THEN
    Result := Machine.RegisterExternalController(ControlSourceHMI);
END_IF

IF NOT ControlSourcePB.Registered THEN
    Result := Machine.RegisterExternalController(ControlSourcePB);
END_IF

ControlSourceHMI.CyclicLogic();
ControlSourcePB.CyclicLogic();

ADSLOGSTR(ADSLOG_MSGTYPE_WARN, 'Lag Monitoring disabled', 'For simulation demo only',);

Initialize := TRUE;
END_METHOD

END_PROGRAM

// ---- GlobalTextList.TcGTLO
TEXTLIST GlobalTextList
  996 = '%3.1f'
  188 = '%d'
  685 = '%s'
  309 = '%S'
  638 = '%x'
  508 = '%X'
  81 = '1'
  902 = '2'
  489 = '3'
  115 = '4'
  268 = '5'
  366 = '6'
  453 = 'A'
  680 = 'Abort'
  8 = 'B'
  122 = 'BAO Jam PE'
  139 = 'Bridge Breaker Down'
  111 = 'Bridge Breaker Up'
  557 = 'C'
  452 = 'Clear'
  276 = 'Disc Level PE'
  217 = 'Downstream Backup PE'
  280 = 'Enabled'
  54 = 'Exit Jam PE'
  316 = 'Fault'
  842 = 'Has Mover'
  944 = 'HMI PB Station'
  744 = 'Hold'
  53 = 'Home'
  551 = 'Hopper Level PE'
  182 = 'Initialized'
  938 = 'M1'
  892 = 'M10'
  219 = 'M11'
  144 = 'M12'
  303 = 'M2'
  38 = 'M3'
  609 = 'M4'
  227 = 'M5'
  875 = 'M6'
  108 = 'M7'
  154 = 'M8'
  216 = 'M9'
  347 = 'MACHINE'
  822 = 'MACHINE STATE CONTROL'
  46 = 'Maintenance'
  904 = 'Manual'
  114 = 'Mover'
  374 = 'Mover Fault'
  899 = 'Movers'
  463 = 'Number of Movers'
  78 = 'Number of Statinon'
  735 = 'Number of Statins'
  915 = 'Number of Stations'
  667 = 'Number of Tracks'
  49 = 'Operational Control Pad'
  880 = 'PowerOK'
  929 = 'Production'
  924 = 'Pushbutton Station'
  181 = 'Reset'
  252 = 'Send Away'
  780 = 'Speed Shift PE'
  77 = 'Start'
  839 = 'State-Machine Pad'
  516 = 'State: %s'
  739 = 'Stations'
  828 = 'Stop'
  806 = 'Suspend'
  386 = 'Tile Count'
  499 = 'Track'
  197 = 'Unhold'
  832 = 'Unsuspend'
  466 = 'Utility'
  785 = 'X'
  984 = 'XPlanar Example Project'
  88 = 'XPlanar Table'
  440 = 'Y'
  313 = 'y'
  438 = 'Z'
END_TEXTLIST

// ---- Machine/VISUs/VisuOjects/V_Control_Xplanar.TcVIS
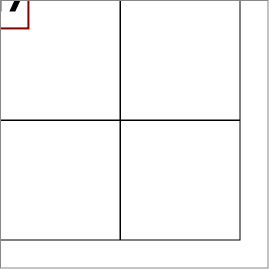
VISUALIZATION V_Control_Xplanar  // 269x269
    Rectangle (0,0 120x120)
    Rectangle (120,0 120x120)
    Rectangle (0,120 120x120)
    Rectangle (120,120 120x120)
    Rectangle (-29,-29 57x57), "M1"
        p3560616238: stMoverVis[1].fPosition_X/2
        p2738717112: (480-stMoverVis[1].fPosition_Y)/2
        p2858320360: stMoverVis[1].fPosition_C
    Rectangle (-29,-29 58x58), "1", invisible if: NOT stStationVis[1].bInit
        p3560616238: stStationVis[1].fPosition_X/2
        p2738717112: (480-stStationVis[1].fPosition_Y)/2
    Rectangle (-29,-29 58x58), "2", invisible if: NOT stStationVis[2].bInit
        p3560616238: stStationVis[2].fPosition_X/2
        p2738717112: (480-stStationVis[2].fPosition_Y)/2
    Rectangle (-29,-29 58x58), "3", invisible if: NOT stStationVis[1].bInit
        p3560616238: stStationVis[3].fPosition_X/2
        p2738717112: (480-stStationVis[3].fPosition_Y)/2
    Rectangle (-29,-29 57x57), "M6"
        p3560616238: stMoverVis[6].fPosition_X/2
        p2738717112: (480-stMoverVis[6].fPosition_Y)/2
        p2858320360: stMoverVis[6].fPosition_C
    Rectangle (-29,-29 57x57), "M5"
        p3560616238: stMoverVis[5].fPosition_X/2
        p2738717112: (480-stMoverVis[5].fPosition_Y)/2
        p2858320360: stMoverVis[5].fPosition_C
    Rectangle (-29,-29 57x57), "M4"
        p3560616238: stMoverVis[4].fPosition_X/2
        p2738717112: (480-stMoverVis[4].fPosition_Y)/2
        p2858320360: stMoverVis[4].fPosition_C
    Rectangle (-29,-29 57x57), "M3"
        p3560616238: stMoverVis[3].fPosition_X/2
        p2738717112: (480-stMoverVis[3].fPosition_Y)/2
        p2858320360: stMoverVis[3].fPosition_C
    Rectangle (-29,-29 57x57), "M2"
        p3560616238: stMoverVis[2].fPosition_X/2
        p2738717112: (480-stMoverVis[2].fPosition_Y)/2
        p2858320360: stMoverVis[2].fPosition_C
    Rectangle (-29,-29 57x57), "M12"
        p3560616238: stMoverVis[12].fPosition_X/2
        p2738717112: (480-stMoverVis[12].fPosition_Y)/2
        p2858320360: stMoverVis[12].fPosition_C
    Rectangle (-29,-29 57x57), "M11"
        p3560616238: stMoverVis[11].fPosition_X/2
        p2738717112: (480-stMoverVis[11].fPosition_Y)/2
        p2858320360: stMoverVis[11].fPosition_C
    Rectangle (-29,-29 57x57), "M10"
        p3560616238: stMoverVis[10].fPosition_X/2
        p2738717112: (480-stMoverVis[10].fPosition_Y)/2
        p2858320360: stMoverVis[10].fPosition_C
    Rectangle (-29,-29 57x57), "M9"
        p3560616238: stMoverVis[9].fPosition_X/2
        p2738717112: (480-stMoverVis[9].fPosition_Y)/2
        p2858320360: stMoverVis[9].fPosition_C
    Rectangle (-29,-29 57x57), "M8"
        p3560616238: stMoverVis[8].fPosition_X/2
        p2738717112: (480-stMoverVis[8].fPosition_Y)/2
        p2858320360: stMoverVis[8].fPosition_C
    Rectangle (-29,-29 57x57), "M7"
        p3560616238: stMoverVis[7].fPosition_X/2
        p2738717112: (480-stMoverVis[7].fPosition_Y)/2
        p2858320360: stMoverVis[7].fPosition_C
END_VISUALIZATION

// ---- Machine/VISUs/VisuOjects/V_MachineModule.TcVIS
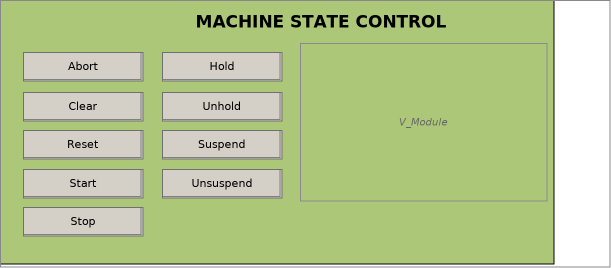
VISUALIZATION V_MachineModule  // 611x268
VAR_IN_OUT
	HMI : ST_PackMLBaseModule_HMI;
END_VAR
    RoundedRectangle (0,-4 554x268)
    Button (23,52 120x29), "Abort"
        OnMouseClick: execute { HMI.Command.State := E_PMLCommand.ePMLCommand_Abort; }
    Button (23,92 120x29), "Clear"
        OnMouseClick: execute { HMI.Command.State := E_PMLCommand.ePMLCommand_Clear; }
    Button (23,130 120x29), "Reset"
        OnMouseClick: execute { HMI.Command.State := E_PMLCommand.ePMLCommand_Reset; }
    Button (23,169 120x29), "Start"
        OnMouseClick: execute { HMI.Command.State := E_PMLCommand.ePMLCommand_Start; }
    Button (23,207 120x29), "Stop"
        OnMouseClick: execute { HMI.Command.State := E_PMLCommand.ePMLCommand_Stop; }
    Button (162,52 120x29), "Hold"
        OnMouseClick: execute { HMI.Command.State := E_PMLCommand.ePMLCommand_Hold; }
    Button (162,92 120x29), "Unhold"
        OnMouseClick: execute { HMI.Command.State := E_PMLCommand.ePMLCommand_Unhold; }
    Button (162,130 120x29), "Suspend"
        OnMouseClick: execute { HMI.Command.State := E_PMLCommand.ePMLCommand_Suspend; }
    Button (162,169 120x29), "Unsuspend"
        OnMouseClick: execute { HMI.Command.State := E_PMLCommand.ePMLCommand_Unsuspend; }
    Frame (300,43 247x158)
        shows V_Module(HMI := HMI)
    Label (31,3 580x37), "MACHINE STATE CONTROL"
END_VISUALIZATION

// ---- Machine/VISUs/VisuOjects/V_Station.TcVIS
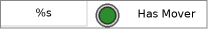
VISUALIZATION V_Station  // 208x29
VAR_IN_OUT
	Station : ST_Station_HMI;
END_VAR
    Textfield (0,0 87x26), "%s", text variable: Station.Status.MoverID
    Lamp1 (92,2 31x27), variable: Station.Status.HasMover, style: Lamp-Lamp1-Green
    Textfield (125,1 83x26), "Has Mover"
END_VISUALIZATION

// ---- Machine/VISUs/V_Main.TcVIS
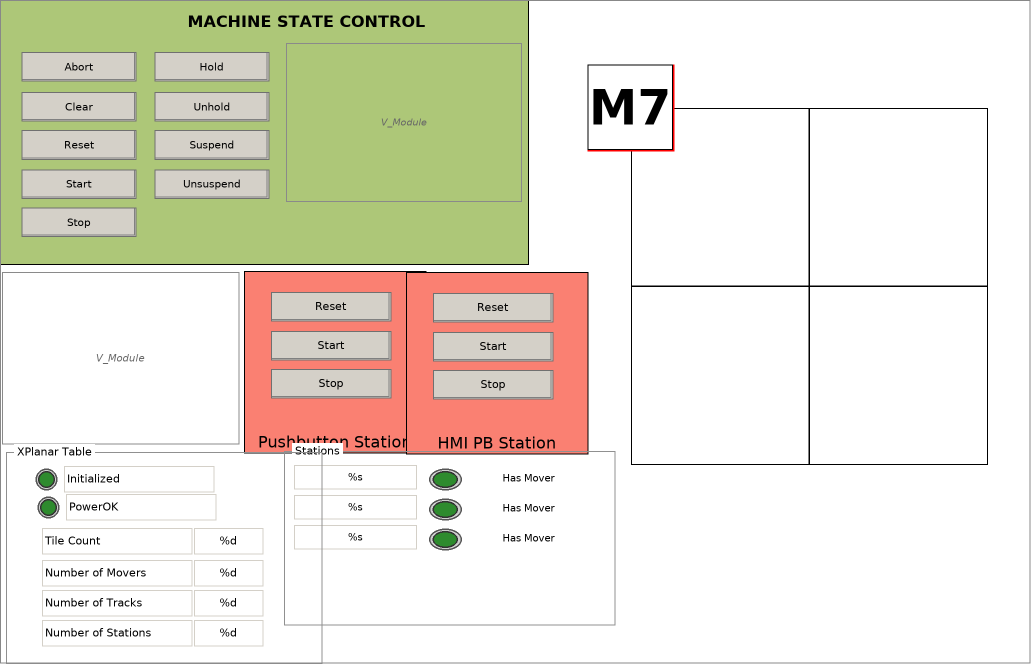
VISUALIZATION V_Main  // 1031x664
    Frame (0,0 583x269)
        shows V_MachineModule(HMI := MAIN.Machine.PackMLBaseModule_HMI)
    Frame (2,272 237x172)
        shows V_Module(HMI := MAIN.Machine.XPlanar.PackMLBaseModule_HMI)
    Group (244,271 156x175)
        RoundedRectangle (0,0 182x182), "Pushbutton Station"
        Button (27,98 120x29), "Stop", input disabled if: not MAIN.ControlSourcePB.MainPMLControl_Simplified.StopPermissive
            tap MAIN.ControlSourcePB.MainPMLControl_Simplified.StopPressed
        Button (27,21 120x29), "Reset", input disabled if: not MAIN.ControlSourcePB.MainPMLControl_Simplified.ResetPermissive
            tap MAIN.ControlSourcePB.MainPMLControl_Simplified.ResetPressed
        Button (27,60 120x29), "Start", input disabled if: not MAIN.ControlSourcePB.MainPMLControl_Simplified.StartPermissive
            tap MAIN.ControlSourcePB.MainPMLControl_Simplified.StartPressed
    Group (406,272 133x175)
        RoundedRectangle (0,0 182x182), "HMI PB Station"
        Button (27,98 120x29), "Stop", input disabled if: not MAIN.ControlSourceHMI.MainPMLControl_Simplified.StopPermissive
            tap MAIN.ControlSourceHMI.MainPMLControl_Simplified.StopPressed
        Button (27,21 120x29), "Reset", input disabled if: not MAIN.ControlSourceHMI.MainPMLControl_Simplified.ResetPermissive
            tap MAIN.ControlSourceHMI.MainPMLControl_Simplified.ResetPressed
        Button (27,60 120x29), "Start", input disabled if: not MAIN.ControlSourceHMI.MainPMLControl_Simplified.StartPermissive
            tap MAIN.ControlSourceHMI.MainPMLControl_Simplified.StartPressed
    Group (284,443 257x219)
        Frame (10,22 293x27)
            shows V_Station(Station := MAIN.Machine.XPlanar.Station1.Station_HMI)
        Frame (10,52 293x27)
            shows V_Station(Station := MAIN.Machine.XPlanar.Station2.Station_HMI)
        Frame (10,82 293x27)
            shows V_Station(Station := MAIN.Machine.XPlanar.Station3.Station_HMI)
        GroupBox (0,0 331x182), "Stations"
    Group (6,444 280x220)
        Lamp1 (28,23 25x25), variable: MAIN.Machine.XPlanar.XPlanarTable.XPlanar_HMI.Status.Initialized, style: Lamp-Lamp1-Green
        Textfield (58,22 150x26), "Initialized"
        Lamp1 (30,51 25x25), variable: MAIN.Machine.XPlanar.XPlanarTable.XPlanar_HMI.Status.PowerOK, style: Lamp-Lamp1-Green
        Textfield (60,50 150x26), "PowerOK"
        Textfield (188,84 69x26), "%d", text variable: MAIN.Machine.XPlanar.XPlanarTable.XPlanar_HMI.Status.TileCount
        Textfield (36,84 150x26), "Tile Count"
        Textfield (188,116 69x26), "%d", text variable: MAIN.Machine.XPlanar.XPlanarTable.XPlanar_HMI.Status.NumberOfMovers
        Textfield (36,116 150x26), "Number of Movers"
        Textfield (188,146 69x26), "%d", text variable: MAIN.Machine.XPlanar.XPlanarTable.XPlanar_HMI.Status.NumberOfTracks
        Textfield (36,146 150x26), "Number of Tracks"
        Textfield (188,176 69x26), "%d", text variable: MAIN.Machine.XPlanar.XPlanarTable.XPlanar_HMI.Status.NumberOfStations
        Textfield (36,176 150x26), "Number of Stations"
        GroupBox (0,0 316x220), "XPlanar Table"
    Frame (631,108 400x400)
        shows V_Control_Xplanar()
END_VISUALIZATION
